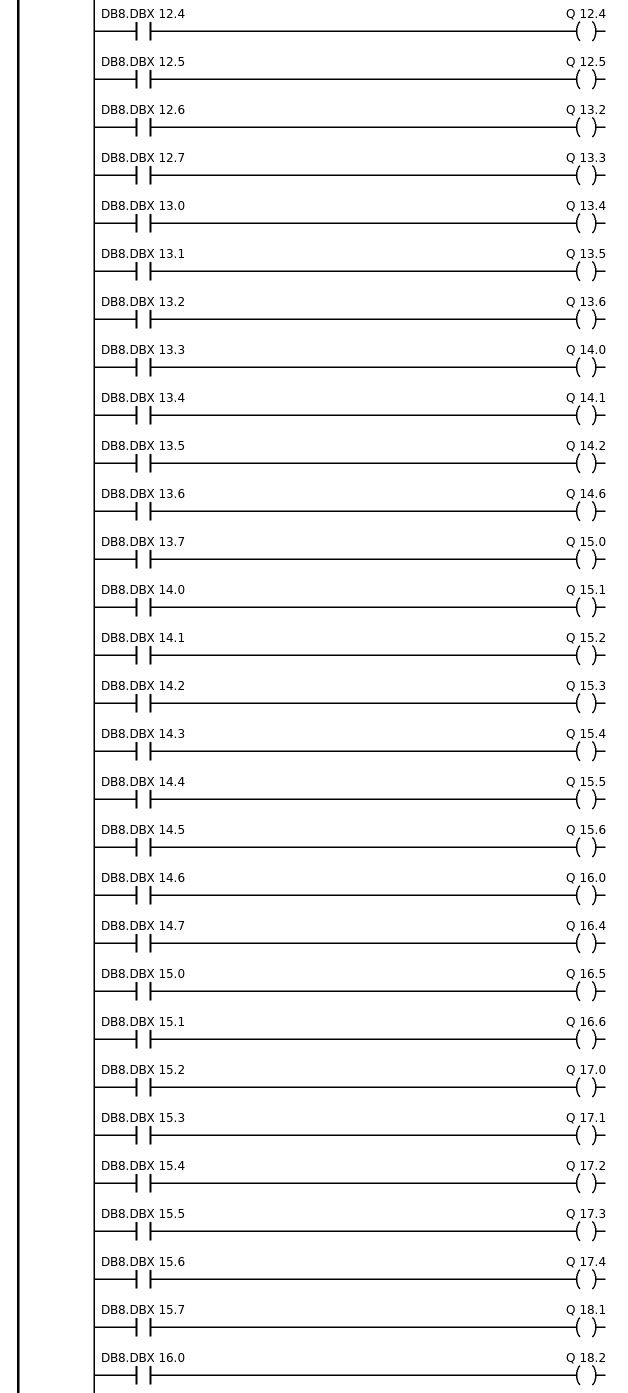
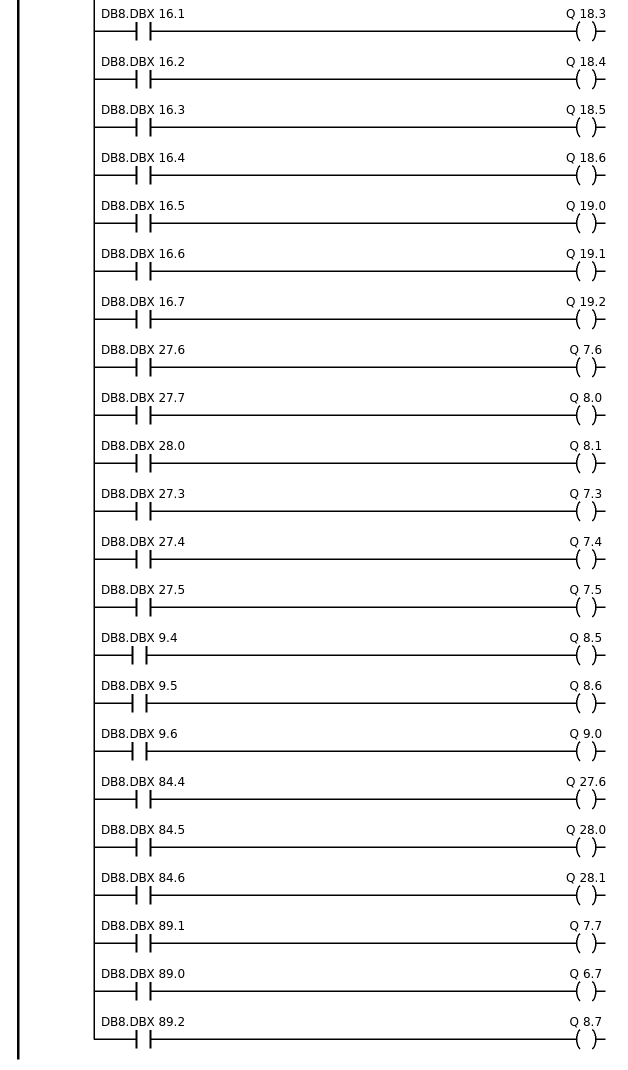
NETWORK
TITLE =
      A     M 0.1;
      =     L 0.0;
      A     L 0.0;
      A     DB8.DBX 26.7;
      =     Q 6.6;
      A     L 0.0;
      A     DB8.DBX 27.0;
      =     Q 7.0;
      A     L 0.0;
      A     DB8.DBX 27.1;
      =     Q 7.1;
      A     L 0.0;
      A     DB8.DBX 27.2;
      =     Q 7.2;
      A     L 0.0;
      A     DB8.DBX 9.1;
      =     Q 8.2;
      A     L 0.0;
      A     DB8.DBX 9.2;
      =     Q 8.3;
      A     L 0.0;
      A     DB8.DBX 9.3;
      =     Q 8.4;
      A     L 0.0;
      A     DB8.DBX 9.7;
      =     Q 9.1;
      A     L 0.0;
      A     DB8.DBX 10.0;
      =     Q 9.2;
      A     L 0.0;
      A     DB8.DBX 10.1;
      =     Q 9.3;
      A     L 0.0;
      A     DB8.DBX 10.2;
      =     Q 9.4;
      A     L 0.0;
      A     DB8.DBX 10.3;
      =     Q 9.5;
      A     L 0.0;
      A     DB8.DBX 10.4;
      =     Q 9.6;
      A     L 0.0;
      A     DB8.DBX 10.5;
      =     Q 10.0;
      A     L 0.0;
      A     DB8.DBX 10.6;
      =     Q 10.1;
      A     L 0.0;
      A     DB8.DBX 10.7;
      =     Q 10.2;
      A     L 0.0;
      A     DB8.DBX 11.0;
      =     Q 10.3;
      A     L 0.0;
      A     DB8.DBX 11.1;
      =     Q 10.4;
      A     L 0.0;
      A     DB8.DBX 11.2;
      =     Q 10.5;
      A     L 0.0;
      A     DB8.DBX 11.3;
      =     Q 10.6;
      A     L 0.0;
      A     DB8.DBX 11.4;
      =     Q 11.0;
      A     L 0.0;
      A     DB8.DBX 11.5;
      =     Q 11.4;
      A     L 0.0;
      A     DB8.DBX 11.6;
      =     Q 11.5;
      A     L 0.0;
      A     DB8.DBX 11.7;
      =     Q 11.6;
      A     L 0.0;
      A     DB8.DBX 12.0;
      =     Q 12.0;
      A     L 0.0;
      A     DB8.DBX 12.1;
      =     Q 12.1;
      A     L 0.0;
      A     DB8.DBX 12.2;
      =     Q 12.2;
      A     L 0.0;
      A     DB8.DBX 12.3;
      =     Q 12.3;
      A     L 0.0;
      A     DB8.DBX 12.4;
      =     Q 12.4;
      A     L 0.0;
      A     DB8.DBX 12.5;
      =     Q 12.5;
      A     L 0.0;
      A     DB8.DBX 12.6;
      =     Q 13.2;
      A     L 0.0;
      A     DB8.DBX 12.7;
      =     Q 13.3;
      A     L 0.0;
      A     DB8.DBX 13.0;
      =     Q 13.4;
      A     L 0.0;
      A     DB8.DBX 13.1;
      =     Q 13.5;
      A     L 0.0;
      A     DB8.DBX 13.2;
      =     Q 13.6;
      A     L 0.0;
      A     DB8.DBX 13.3;
      =     Q 14.0;
      A     L 0.0;
      A     DB8.DBX 13.4;
      =     Q 14.1;
      A     L 0.0;
      A     DB8.DBX 13.5;
      =     Q 14.2;
      A     L 0.0;
      A     DB8.DBX 13.6;
      =     Q 14.6;
      A     L 0.0;
      A     DB8.DBX 13.7;
      =     Q 15.0;
      A     L 0.0;
      A     DB8.DBX 14.0;
      =     Q 15.1;
      A     L 0.0;
      A     DB8.DBX 14.1;
      =     Q 15.2;
      A     L 0.0;
      A     DB8.DBX 14.2;
      =     Q 15.3;
      A     L 0.0;
      A     DB8.DBX 14.3;
      =     Q 15.4;
      A     L 0.0;
      A     DB8.DBX 14.4;
      =     Q 15.5;
      A     L 0.0;
      A     DB8.DBX 14.5;
      =     Q 15.6;
      A     L 0.0;
      A     DB8.DBX 14.6;
      =     Q 16.0;
      A     L 0.0;
      A     DB8.DBX 14.7;
      =     Q 16.4;
      A     L 0.0;
      A     DB8.DBX 15.0;
      =     Q 16.5;
      A     L 0.0;
      A     DB8.DBX 15.1;
      =     Q 16.6;
      A     L 0.0;
      A     DB8.DBX 15.2;
      =     Q 17.0;
      A     L 0.0;
      A     DB8.DBX 15.3;
      =     Q 17.1;
      A     L 0.0;
      A     DB8.DBX 15.4;
      =     Q 17.2;
      A     L 0.0;
      A     DB8.DBX 15.5;
      =     Q 17.3;
      A     L 0.0;
      A     DB8.DBX 15.6;
      =     Q 17.4;
      A     L 0.0;
      A     DB8.DBX 15.7;
      =     Q 18.1;
      A     L 0.0;
      A     DB8.DBX 16.0;
      =     Q 18.2;
      A     L 0.0;
      A     DB8.DBX 16.1;
      =     Q 18.3;
      A     L 0.0;
      A     DB8.DBX 16.2;
      =     Q 18.4;
      A     L 0.0;
      A     DB8.DBX 16.3;
      =     Q 18.5;
      A     L 0.0;
      A     DB8.DBX 16.4;
      =     Q 18.6;
      A     L 0.0;
      A     DB8.DBX 16.5;
      =     Q 19.0;
      A     L 0.0;
      A     DB8.DBX 16.6;
      =     Q 19.1;
      A     L 0.0;
      A     DB8.DBX 16.7;
      =     Q 19.2;
      A     L 0.0;
      A     DB8.DBX 27.6;
      =     Q 7.6;
      A     L 0.0;
      A     DB8.DBX 27.7;
      =     Q 8.0;
      A     L 0.0;
      A     DB8.DBX 28.0;
      =     Q 8.1;
      A     L 0.0;
      A     DB8.DBX 27.3;
      =     Q 7.3;
      A     L 0.0;
      A     DB8.DBX 27.4;
      =     Q 7.4;
      A     L 0.0;
      A     DB8.DBX 27.5;
      =     Q 7.5;
      A     L 0.0;
      A     DB8.DBX 9.4;
      =     Q 8.5;
      A     L 0.0;
      A     DB8.DBX 9.5;
      =     Q 8.6;
      A     L 0.0;
      A     DB8.DBX 9.6;
      =     Q 9.0;
      A     L 0.0;
      A     DB8.DBX 84.4;
      =     Q 27.6;
      A     L 0.0;
      A     DB8.DBX 84.5;
      =     Q 28.0;
      A     L 0.0;
      A     DB8.DBX 84.6;
      =     Q 28.1;
      A     L 0.0;
      A     DB8.DBX 89.1;
      =     Q 7.7;
      A     L 0.0;
      A     DB8.DBX 89.0;
      =     Q 6.7;
      A     L 0.0;
      A     DB8.DBX 89.2;
      =     Q 8.7;
END_FUNCTION

FUNCTION FC 7 : VOID
AUTHOR : Arun_Ram
VERSION : 0.1
BEGIN
// (block stored without names or comments; labels and parameter names are numbered)
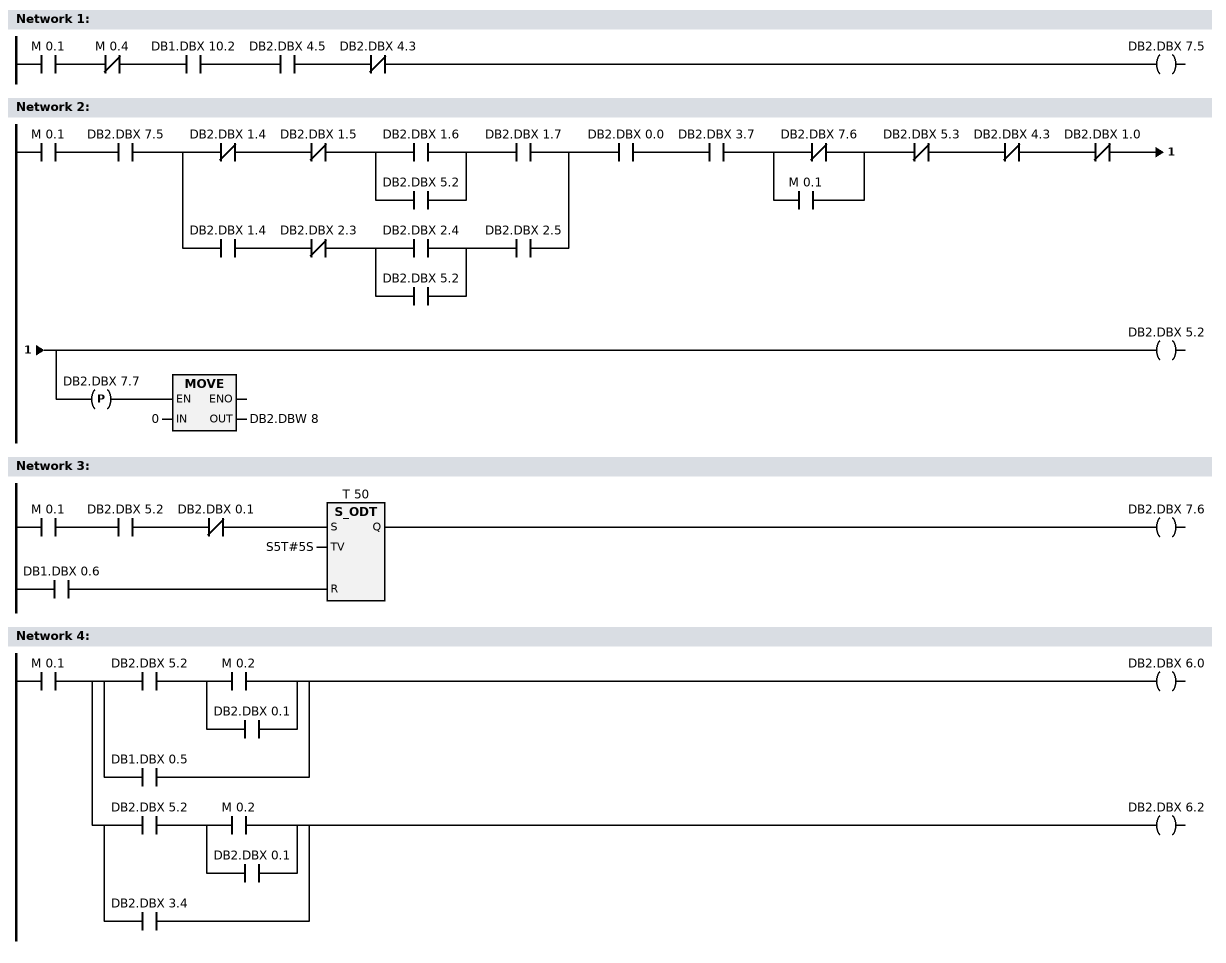
NETWORK
TITLE =
      A     M 0.1;
      AN    M 0.4;
      A     DB1.DBX 10.2;
      A     DB2.DBX 4.5;
      AN    DB2.DBX 4.3;
      =     DB2.DBX 7.5;
NETWORK
TITLE =
      A     M 0.1;
      A     DB2.DBX 7.5;
      A(;
      AN    DB2.DBX 1.4;
      AN    DB2.DBX 1.5;
      A(;
      O     DB2.DBX 1.6;
      O     DB2.DBX 5.2;
      );
      A     DB2.DBX 1.7;
      O;
      A     DB2.DBX 1.4;
      AN    DB2.DBX 2.3;
      A(;
      O     DB2.DBX 2.4;
      O     DB2.DBX 5.2;
      );
      A     DB2.DBX 2.5;
      );
      A     DB2.DBX 0.0;
      A     DB2.DBX 3.7;
      A(;
      ON    DB2.DBX 7.6;
      O     M 0.1;
      );
      AN    DB2.DBX 5.3;
      AN    DB2.DBX 4.3;
      AN    DB2.DBX 1.0;
      =     L 0.0;
      A     L 0.0;
      BLD   102;
      =     DB2.DBX 5.2;
      A     L 0.0;
      FP    DB2.DBX 7.7;
      JNB   M001;
      L     0;
      T     DB2.DBW 8;
M001: NOP   0;
NETWORK
TITLE =
      A     M 0.1;
      A     DB2.DBX 5.2;
      AN    DB2.DBX 0.1;
      L     S5T#5S;
      SD    T 50;
      A     DB1.DBX 0.6;
      R     T 50;
      NOP   0;
      NOP   0;
      A     T 50;
      =     DB2.DBX 7.6;
NETWORK
TITLE =
      A     M 0.1;
      =     L 0.0;
      A     L 0.0;
      A(;
      A     DB2.DBX 5.2;
      A(;
      O     M 0.2;
      O     DB2.DBX 0.1;
      );
      O     DB1.DBX 0.5;
      );
      =     DB2.DBX 6.0;
      A     L 0.0;
      A(;
      A     DB2.DBX 5.2;
      A(;
      O     M 0.2;
      O     DB2.DBX 0.1;
      );
      O     DB2.DBX 3.4;
      );
      =     DB2.DBX 6.2;
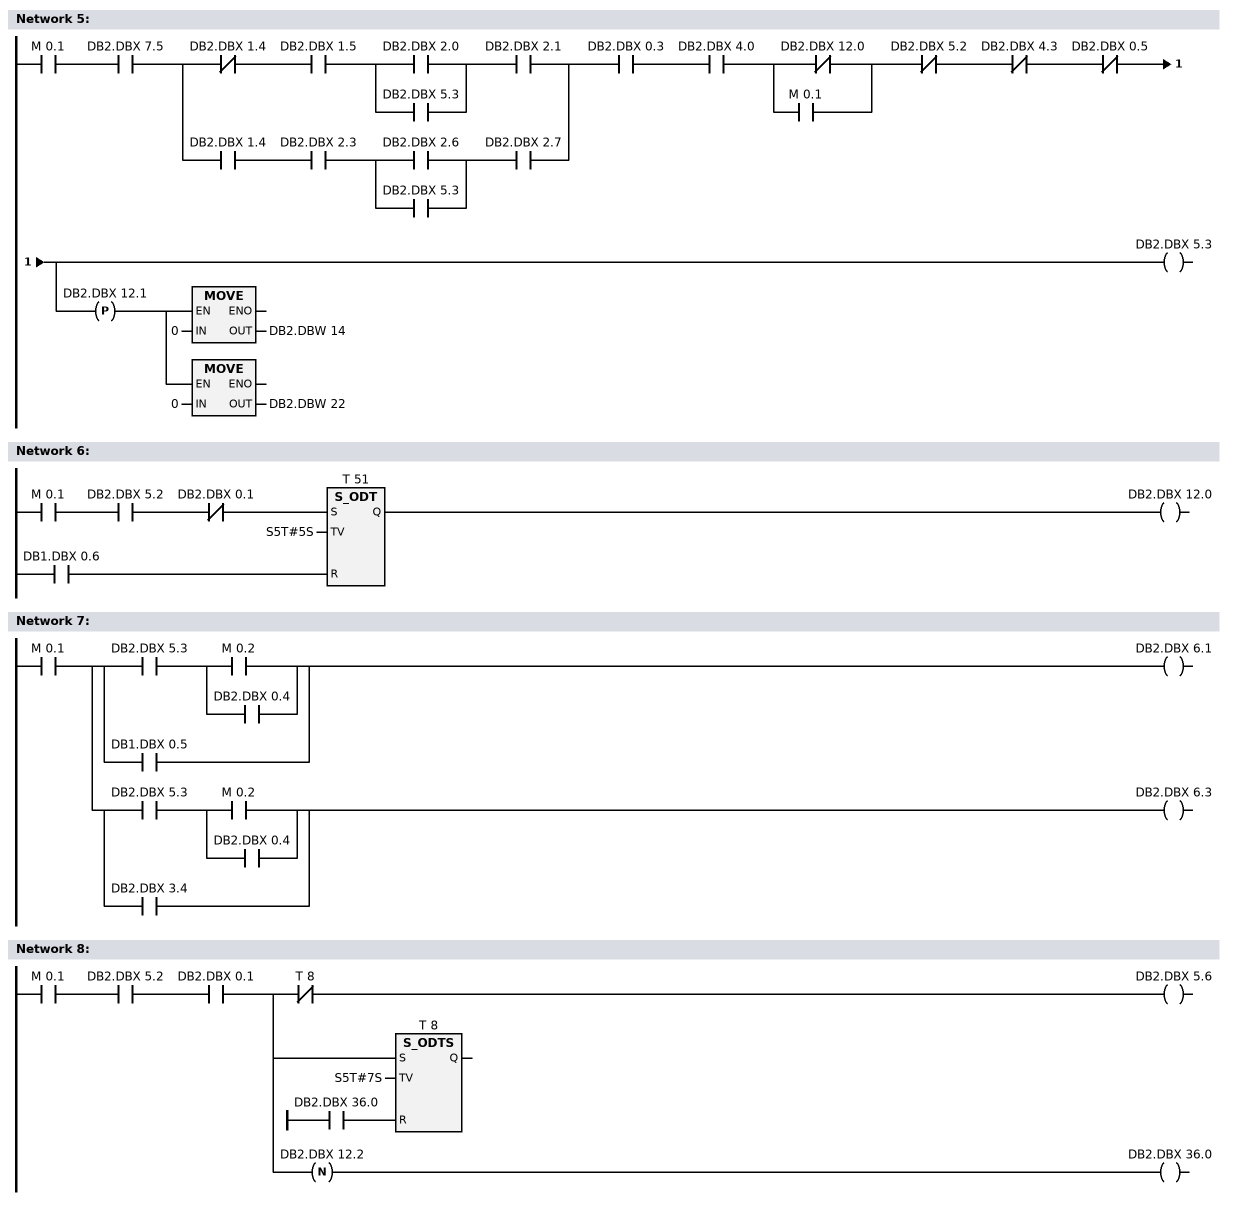
NETWORK
TITLE =
      A     M 0.1;
      A     DB2.DBX 7.5;
      A(;
      AN    DB2.DBX 1.4;
      A     DB2.DBX 1.5;
      A(;
      O     DB2.DBX 2.0;
      O     DB2.DBX 5.3;
      );
      A     DB2.DBX 2.1;
      O;
      A     DB2.DBX 1.4;
      A     DB2.DBX 2.3;
      A(;
      O     DB2.DBX 2.6;
      O     DB2.DBX 5.3;
      );
      A     DB2.DBX 2.7;
      );
      A     DB2.DBX 0.3;
      A     DB2.DBX 4.0;
      A(;
      ON    DB2.DBX 12.0;
      O     M 0.1;
      );
      AN    DB2.DBX 5.2;
      AN    DB2.DBX 4.3;
      AN    DB2.DBX 0.5;
      =     L 0.0;
      A     L 0.0;
      BLD   102;
      =     DB2.DBX 5.3;
      A     L 0.0;
      FP    DB2.DBX 12.1;
      =     L 0.1;
      A     L 0.1;
      JNB   M002;
      L     0;
      T     DB2.DBW 14;
M002: NOP   0;
      A     L 0.1;
      JNB   M003;
      L     0;
      T     DB2.DBW 22;
M003: NOP   0;
NETWORK
TITLE =
      A     M 0.1;
      A     DB2.DBX 5.2;
      AN    DB2.DBX 0.1;
      L     S5T#5S;
      SD    T 51;
      A     DB1.DBX 0.6;
      R     T 51;
      NOP   0;
      NOP   0;
      A     T 51;
      =     DB2.DBX 12.0;
NETWORK
TITLE =
      A     M 0.1;
      =     L 0.0;
      A     L 0.0;
      A(;
      A     DB2.DBX 5.3;
      A(;
      O     M 0.2;
      O     DB2.DBX 0.4;
      );
      O     DB1.DBX 0.5;
      );
      =     DB2.DBX 6.1;
      A     L 0.0;
      A(;
      A     DB2.DBX 5.3;
      A(;
      O     M 0.2;
      O     DB2.DBX 0.4;
      );
      O     DB2.DBX 3.4;
      );
      =     DB2.DBX 6.3;
NETWORK
TITLE =
      A     M 0.1;
      A     DB2.DBX 5.2;
      A     DB2.DBX 0.1;
      =     L 0.0;
      A     L 0.0;
      AN    T 8;
      =     DB2.DBX 5.6;
      A     L 0.0;
      L     S5T#7S;
      SS    T 8;
      A     DB2.DBX 36.0;
      R     T 8;
      NOP   0;
      NOP   0;
      NOP   0;
      A     L 0.0;
      FN    DB2.DBX 12.2;
      =     DB2.DBX 36.0;
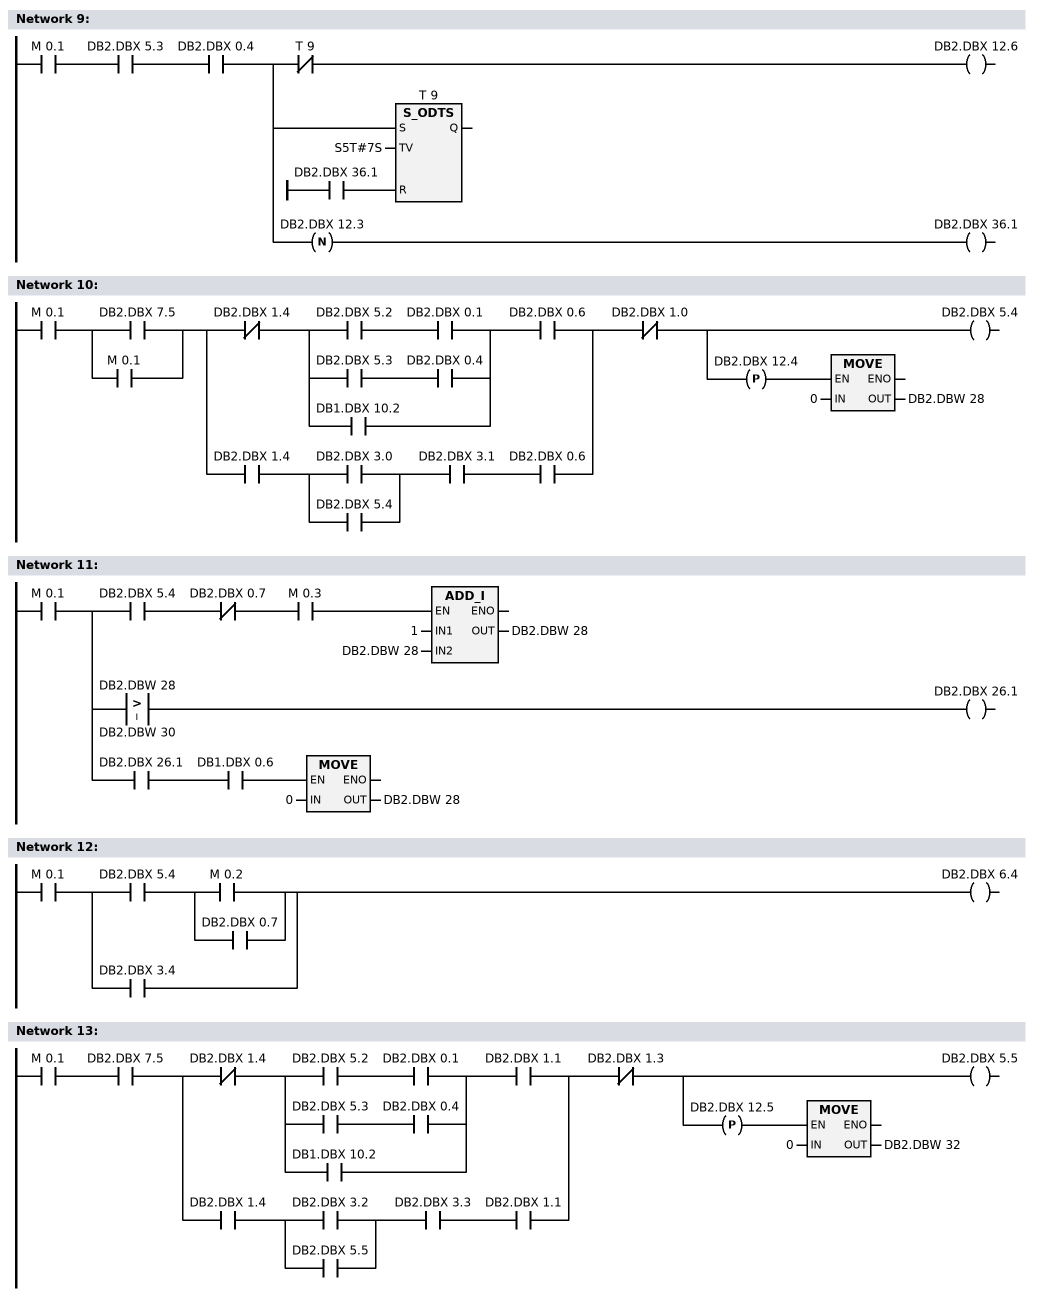
NETWORK
TITLE =
      A     M 0.1;
      A     DB2.DBX 5.3;
      A     DB2.DBX 0.4;
      =     L 0.0;
      A     L 0.0;
      AN    T 9;
      =     DB2.DBX 12.6;
      A     L 0.0;
      L     S5T#7S;
      SS    T 9;
      A     DB2.DBX 36.1;
      R     T 9;
      NOP   0;
      NOP   0;
      NOP   0;
      A     L 0.0;
      FN    DB2.DBX 12.3;
      =     DB2.DBX 36.1;
NETWORK
TITLE =
      A     M 0.1;
      A(;
      O     DB2.DBX 7.5;
      O     M 0.1;
      );
      A(;
      AN    DB2.DBX 1.4;
      A(;
      A     DB2.DBX 5.2;
      A     DB2.DBX 0.1;
      O;
      A     DB2.DBX 5.3;
      A     DB2.DBX 0.4;
      O     DB1.DBX 10.2;
      );
      A     DB2.DBX 0.6;
      O;
      A     DB2.DBX 1.4;
      A(;
      O     DB2.DBX 3.0;
      O     DB2.DBX 5.4;
      );
      A     DB2.DBX 3.1;
      A     DB2.DBX 0.6;
      );
      AN    DB2.DBX 1.0;
      =     L 0.0;
      A     L 0.0;
      BLD   102;
      =     DB2.DBX 5.4;
      A     L 0.0;
      FP    DB2.DBX 12.4;
      JNB   M004;
      L     0;
      T     DB2.DBW 28;
M004: NOP   0;
NETWORK
TITLE =
      A     M 0.1;
      =     L 0.0;
      A     L 0.0;
      A     DB2.DBX 5.4;
      AN    DB2.DBX 0.7;
      A     M 0.3;
      JNB   M005;
      L     1;
      L     DB2.DBW 28;
      +I;
      T     DB2.DBW 28;
M005: NOP   0;
      A     L 0.0;
      A(;
      L     DB2.DBW 28;
      L     DB2.DBW 30;
      >I;
      );
      =     DB2.DBX 26.1;
      A     L 0.0;
      A     DB2.DBX 26.1;
      A     DB1.DBX 0.6;
      JNB   M006;
      L     0;
      T     DB2.DBW 28;
M006: NOP   0;
NETWORK
TITLE =
      A     M 0.1;
      A(;
      A     DB2.DBX 5.4;
      A(;
      O     M 0.2;
      O     DB2.DBX 0.7;
      );
      O     DB2.DBX 3.4;
      );
      =     DB2.DBX 6.4;
NETWORK
TITLE =
      A     M 0.1;
      A     DB2.DBX 7.5;
      A(;
      AN    DB2.DBX 1.4;
      A(;
      A     DB2.DBX 5.2;
      A     DB2.DBX 0.1;
      O;
      A     DB2.DBX 5.3;
      A     DB2.DBX 0.4;
      O     DB1.DBX 10.2;
      );
      A     DB2.DBX 1.1;
      O;
      A     DB2.DBX 1.4;
      A(;
      O     DB2.DBX 3.2;
      O     DB2.DBX 5.5;
      );
      A     DB2.DBX 3.3;
      A     DB2.DBX 1.1;
      );
      AN    DB2.DBX 1.3;
      =     L 0.0;
      A     L 0.0;
      BLD   102;
      =     DB2.DBX 5.5;
      A     L 0.0;
      FP    DB2.DBX 12.5;
      JNB   M007;
      L     0;
      T     DB2.DBW 32;
M007: NOP   0;
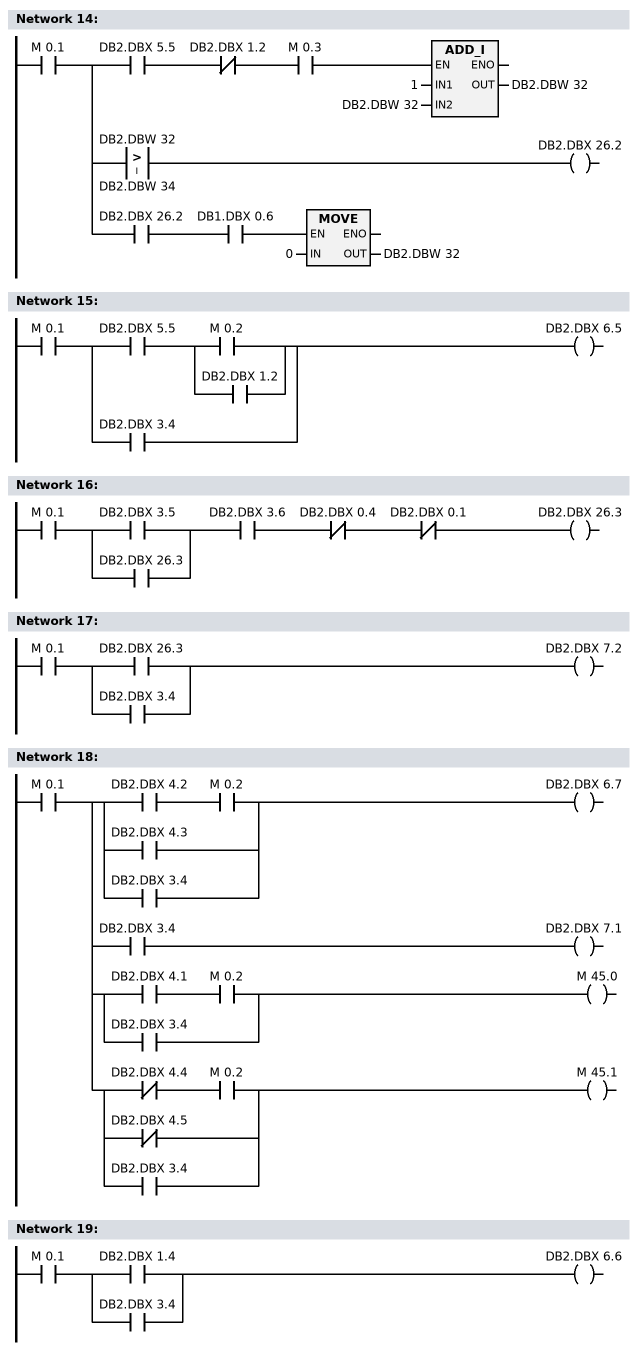
NETWORK
TITLE =
      A     M 0.1;
      =     L 0.0;
      A     L 0.0;
      A     DB2.DBX 5.5;
      AN    DB2.DBX 1.2;
      A     M 0.3;
      JNB   M008;
      L     1;
      L     DB2.DBW 32;
      +I;
      T     DB2.DBW 32;
M008: NOP   0;
      A     L 0.0;
      A(;
      L     DB2.DBW 32;
      L     DB2.DBW 34;
      >I;
      );
      =     DB2.DBX 26.2;
      A     L 0.0;
      A     DB2.DBX 26.2;
      A     DB1.DBX 0.6;
      JNB   M009;
      L     0;
      T     DB2.DBW 32;
M009: NOP   0;
NETWORK
TITLE =
      A     M 0.1;
      A(;
      A     DB2.DBX 5.5;
      A(;
      O     M 0.2;
      O     DB2.DBX 1.2;
      );
      O     DB2.DBX 3.4;
      );
      =     DB2.DBX 6.5;
NETWORK
TITLE =
      A     M 0.1;
      A(;
      O     DB2.DBX 3.5;
      O     DB2.DBX 26.3;
      );
      A     DB2.DBX 3.6;
      AN    DB2.DBX 0.4;
      AN    DB2.DBX 0.1;
      =     DB2.DBX 26.3;
NETWORK
TITLE =
      A     M 0.1;
      A(;
      O     DB2.DBX 26.3;
      O     DB2.DBX 3.4;
      );
      =     DB2.DBX 7.2;
NETWORK
TITLE =
      A     M 0.1;
      =     L 0.0;
      A     L 0.0;
      A(;
      A     DB2.DBX 4.2;
      A     M 0.2;
      O     DB2.DBX 4.3;
      O     DB2.DBX 3.4;
      );
      =     DB2.DBX 6.7;
      A     L 0.0;
      A     DB2.DBX 3.4;
      =     DB2.DBX 7.1;
      A     L 0.0;
      A(;
      A     DB2.DBX 4.1;
      A     M 0.2;
      O     DB2.DBX 3.4;
      );
      =     M 45.0;
      A     L 0.0;
      A(;
      AN    DB2.DBX 4.4;
      A     M 0.2;
      ON    DB2.DBX 4.5;
      O     DB2.DBX 3.4;
      );
      =     M 45.1;
NETWORK
TITLE =
      A     M 0.1;
      A(;
      O     DB2.DBX 1.4;
      O     DB2.DBX 3.4;
      );
      =     DB2.DBX 6.6;
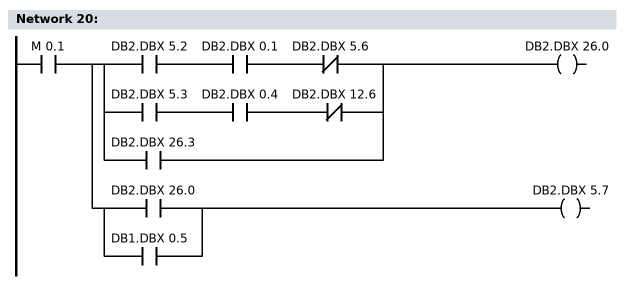
NETWORK
TITLE =
      A     M 0.1;
      =     L 0.0;
      A     L 0.0;
      A(;
      A     DB2.DBX 5.2;
      A     DB2.DBX 0.1;
      AN    DB2.DBX 5.6;
      O;
      A     DB2.DBX 5.3;
      A     DB2.DBX 0.4;
      AN    DB2.DBX 12.6;
      O     DB2.DBX 26.3;
      );
      =     DB2.DBX 26.0;
      A     L 0.0;
      A(;
      O     DB2.DBX 26.0;
      O     DB1.DBX 0.5;
      );
      =     DB2.DBX 5.7;
END_FUNCTION

FUNCTION FC 8 : VOID
AUTHOR : Arun_Ram
VERSION : 0.1
BEGIN
// (block stored without names or comments; labels and parameter names are numbered)
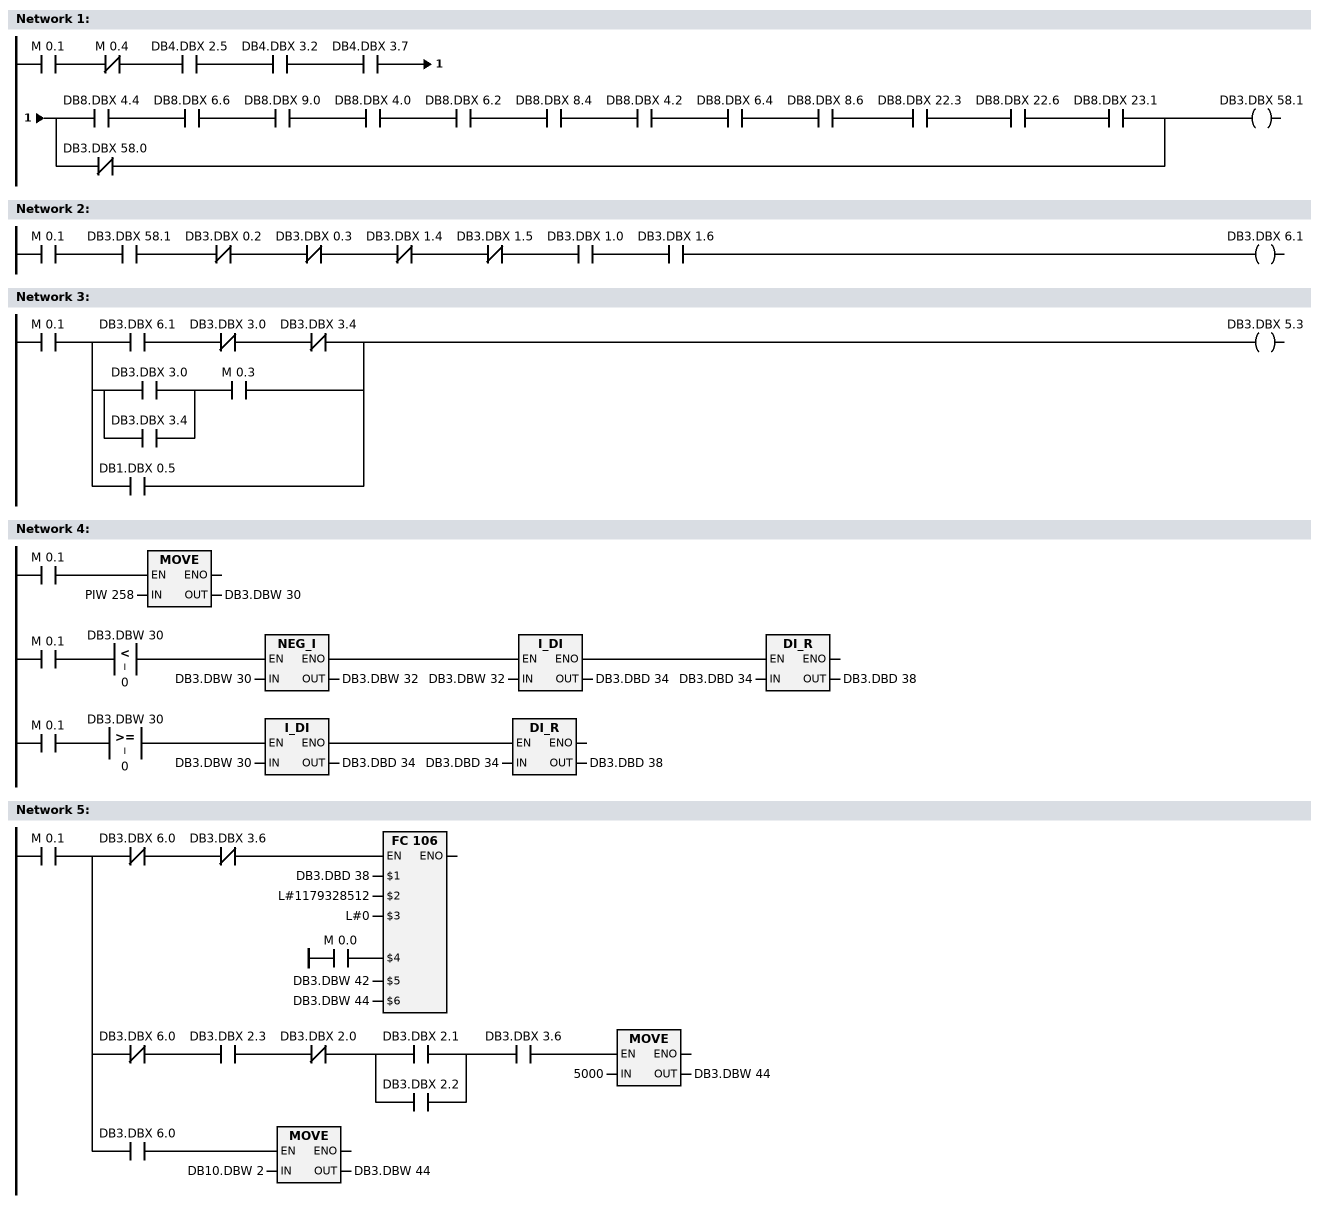
NETWORK
TITLE =
      A     M 0.1;
      AN    M 0.4;
      A     DB4.DBX 2.5;
      A     DB4.DBX 3.2;
      A     DB4.DBX 3.7;
      A(;
      A     DB8.DBX 4.4;
      A     DB8.DBX 6.6;
      A     DB8.DBX 9.0;
      A     DB8.DBX 4.0;
      A     DB8.DBX 6.2;
      A     DB8.DBX 8.4;
      A     DB8.DBX 4.2;
      A     DB8.DBX 6.4;
      A     DB8.DBX 8.6;
      A     DB8.DBX 22.3;
      A     DB8.DBX 22.6;
      A     DB8.DBX 23.1;
      ON    DB3.DBX 58.0;
      );
      =     DB3.DBX 58.1;
NETWORK
TITLE =
      A     M 0.1;
      A     DB3.DBX 58.1;
      AN    DB3.DBX 0.2;
      AN    DB3.DBX 0.3;
      AN    DB3.DBX 1.4;
      AN    DB3.DBX 1.5;
      A     DB3.DBX 1.0;
      A     DB3.DBX 1.6;
      =     DB3.DBX 6.1;
NETWORK
TITLE =
      A     M 0.1;
      A(;
      A     DB3.DBX 6.1;
      AN    DB3.DBX 3.0;
      AN    DB3.DBX 3.4;
      O;
      A(;
      O     DB3.DBX 3.0;
      O     DB3.DBX 3.4;
      );
      A     M 0.3;
      O     DB1.DBX 0.5;
      );
      =     DB3.DBX 5.3;
NETWORK
TITLE =
      A     M 0.1;
      =     L 0.0;
      A     L 0.0;
      JNB   M001;
      L     PIW 258;
      T     DB3.DBW 30;
M001: NOP   0;
      A(;
      A(;
      A     L 0.0;
      A(;
      L     DB3.DBW 30;
      L     0;
      <I;
      );
      JNB   M002;
      L     DB3.DBW 30;
      NEGI;
      T     DB3.DBW 32;
      AN    OV;
      SAVE;
      CLR;
M002: A     BR;
      );
      JNB   M003;
      L     DB3.DBW 32;
      ITD;
      T     DB3.DBD 34;
      SET;
      SAVE;
      CLR;
M003: A     BR;
      );
      JNB   M004;
      L     DB3.DBD 34;
      DTR;
      T     DB3.DBD 38;
M004: NOP   0;
      A(;
      A     L 0.0;
      A(;
      L     DB3.DBW 30;
      L     0;
      >=I;
      );
      JNB   M005;
      L     DB3.DBW 30;
      ITD;
      T     DB3.DBD 34;
      SET;
      SAVE;
      CLR;
M005: A     BR;
      );
      JNB   M006;
      L     DB3.DBD 34;
      DTR;
      T     DB3.DBD 38;
M006: NOP   0;
NETWORK
TITLE =
      A     M 0.1;
      =     L 0.0;
      A     M 0.0;
      =     L 0.1;
      BLD   103;
      A     L 0.0;
      AN    DB3.DBX 6.0;
      AN    DB3.DBX 3.6;
      JNB   M007;
      CALL  FC 106 (
           $1                       := DB3.DBD 38,
           $2                       := L#1179328512,
           $3                       := L#0,
           $4                       := L 0.1,
           $5                       := DB3.DBW 42,
           $6                       := DB3.DBW 44);
M007: NOP   0;
      A     L 0.0;
      AN    DB3.DBX 6.0;
      A     DB3.DBX 2.3;
      AN    DB3.DBX 2.0;
      A(;
      O     DB3.DBX 2.1;
      O     DB3.DBX 2.2;
      );
      A     DB3.DBX 3.6;
      JNB   M008;
      L     5000;
      T     DB3.DBW 44;
M008: NOP   0;
      A     L 0.0;
      A     DB3.DBX 6.0;
      JNB   M009;
      L     DB10.DBW 2;
      T     DB3.DBW 44;
M009: NOP   0;
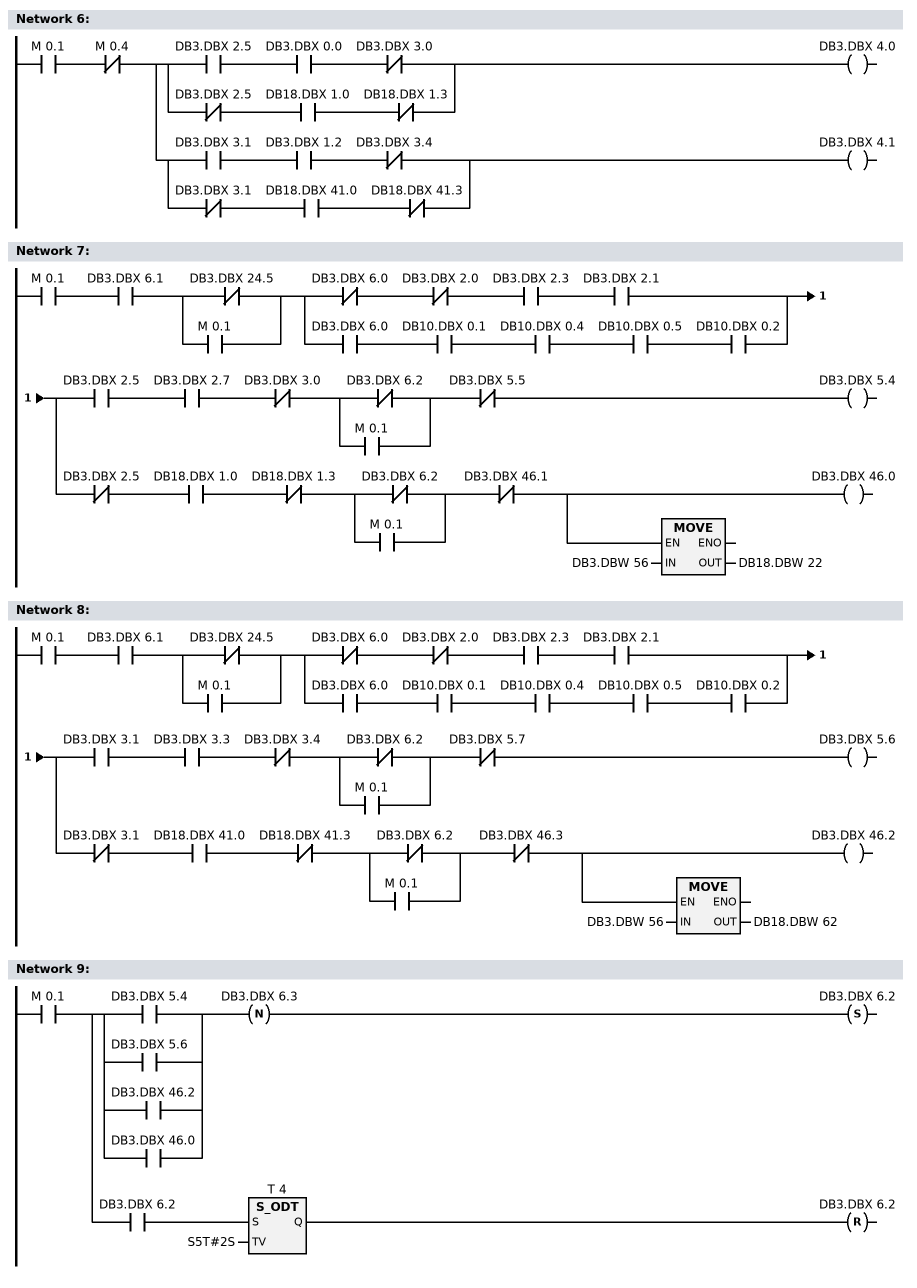
NETWORK
TITLE =
      A     M 0.1;
      AN    M 0.4;
      =     L 0.0;
      A     L 0.0;
      A(;
      A     DB3.DBX 2.5;
      A     DB3.DBX 0.0;
      AN    DB3.DBX 3.0;
      O;
      AN    DB3.DBX 2.5;
      A     DB18.DBX 1.0;
      AN    DB18.DBX 1.3;
      );
      =     DB3.DBX 4.0;
      A     L 0.0;
      A(;
      A     DB3.DBX 3.1;
      A     DB3.DBX 1.2;
      AN    DB3.DBX 3.4;
      O;
      AN    DB3.DBX 3.1;
      A     DB18.DBX 41.0;
      AN    DB18.DBX 41.3;
      );
      =     DB3.DBX 4.1;
NETWORK
TITLE =
      A     M 0.1;
      A     DB3.DBX 6.1;
      A(;
      ON    DB3.DBX 24.5;
      O     M 0.1;
      );
      A(;
      AN    DB3.DBX 6.0;
      AN    DB3.DBX 2.0;
      A     DB3.DBX 2.3;
      A     DB3.DBX 2.1;
      O;
      A     DB3.DBX 6.0;
      A     DB10.DBX 0.1;
      A     DB10.DBX 0.4;
      A     DB10.DBX 0.5;
      A     DB10.DBX 0.2;
      );
      =     L 0.0;
      A     L 0.0;
      A     DB3.DBX 2.5;
      A     DB3.DBX 2.7;
      AN    DB3.DBX 3.0;
      A(;
      ON    DB3.DBX 6.2;
      O     M 0.1;
      );
      AN    DB3.DBX 5.5;
      =     DB3.DBX 5.4;
      A     L 0.0;
      AN    DB3.DBX 2.5;
      A     DB18.DBX 1.0;
      AN    DB18.DBX 1.3;
      A(;
      ON    DB3.DBX 6.2;
      O     M 0.1;
      );
      AN    DB3.DBX 46.1;
      =     L 0.1;
      A     L 0.1;
      BLD   102;
      =     DB3.DBX 46.0;
      A     L 0.1;
      JNB   M010;
      L     DB3.DBW 56;
      T     DB18.DBW 22;
M010: NOP   0;
NETWORK
TITLE =
      A     M 0.1;
      A     DB3.DBX 6.1;
      A(;
      ON    DB3.DBX 24.5;
      O     M 0.1;
      );
      A(;
      AN    DB3.DBX 6.0;
      AN    DB3.DBX 2.0;
      A     DB3.DBX 2.3;
      A     DB3.DBX 2.1;
      O;
      A     DB3.DBX 6.0;
      A     DB10.DBX 0.1;
      A     DB10.DBX 0.4;
      A     DB10.DBX 0.5;
      A     DB10.DBX 0.2;
      );
      =     L 0.0;
      A     L 0.0;
      A     DB3.DBX 3.1;
      A     DB3.DBX 3.3;
      AN    DB3.DBX 3.4;
      A(;
      ON    DB3.DBX 6.2;
      O     M 0.1;
      );
      AN    DB3.DBX 5.7;
      =     DB3.DBX 5.6;
      A     L 0.0;
      AN    DB3.DBX 3.1;
      A     DB18.DBX 41.0;
      AN    DB18.DBX 41.3;
      A(;
      ON    DB3.DBX 6.2;
      O     M 0.1;
      );
      AN    DB3.DBX 46.3;
      =     L 0.1;
      A     L 0.1;
      BLD   102;
      =     DB3.DBX 46.2;
      A     L 0.1;
      JNB   M011;
      L     DB3.DBW 56;
      T     DB18.DBW 62;
M011: NOP   0;
NETWORK
TITLE =
      A     M 0.1;
      =     L 0.0;
      A     L 0.0;
      A(;
      O     DB3.DBX 5.4;
      O     DB3.DBX 5.6;
      O     DB3.DBX 46.2;
      O     DB3.DBX 46.0;
      );
      FN    DB3.DBX 6.3;
      S     DB3.DBX 6.2;
      A     L 0.0;
      A     DB3.DBX 6.2;
      L     S5T#2S;
      SD    T 4;
      NOP   0;
      NOP   0;
      NOP   0;
      A     T 4;
      R     DB3.DBX 6.2;
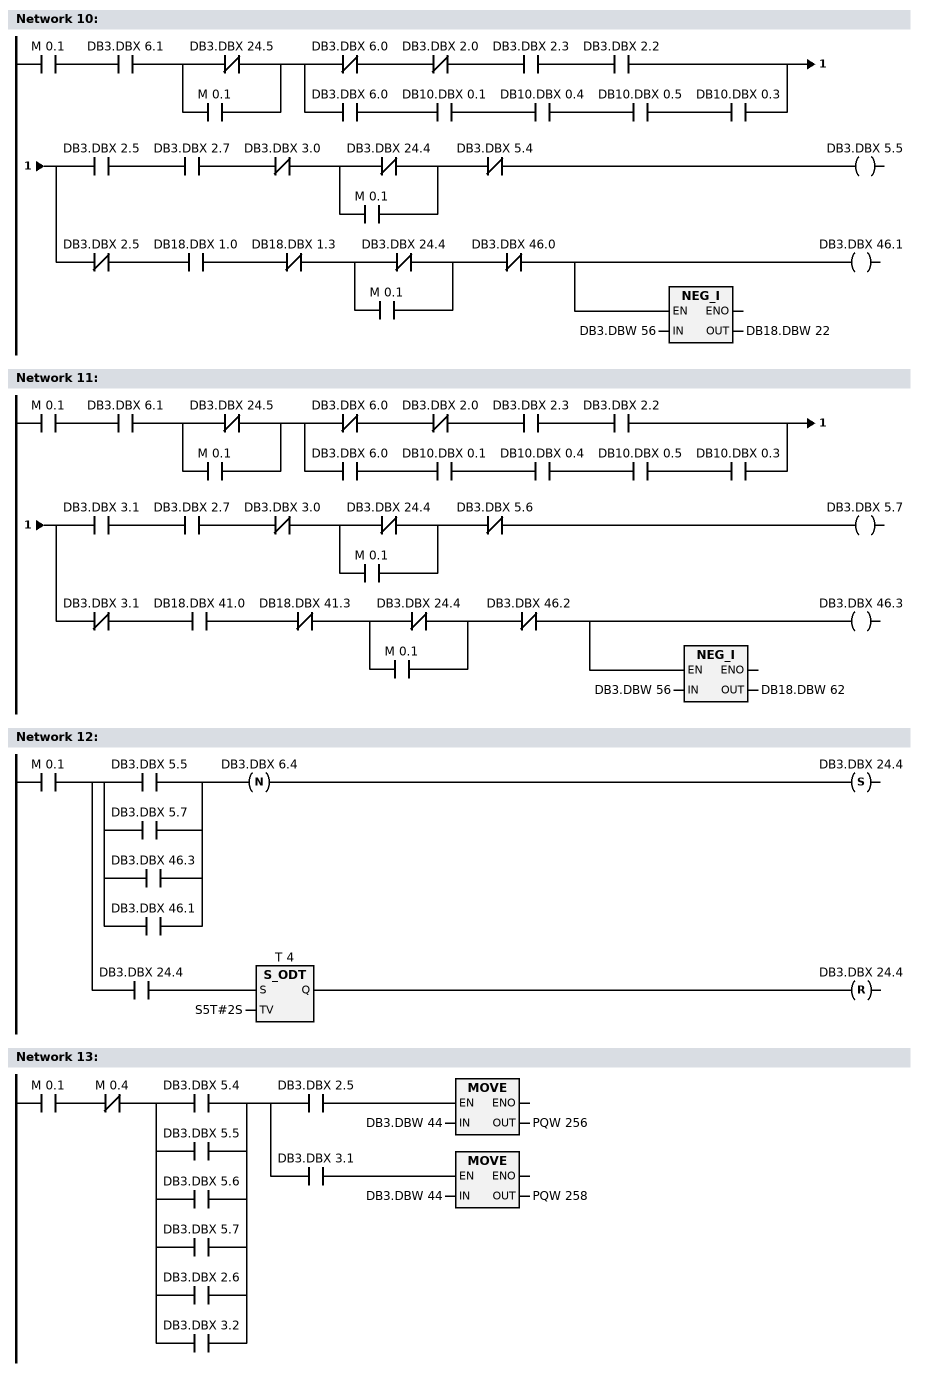
NETWORK
TITLE =
      A     M 0.1;
      A     DB3.DBX 6.1;
      A(;
      ON    DB3.DBX 24.5;
      O     M 0.1;
      );
      A(;
      AN    DB3.DBX 6.0;
      AN    DB3.DBX 2.0;
      A     DB3.DBX 2.3;
      A     DB3.DBX 2.2;
      O;
      A     DB3.DBX 6.0;
      A     DB10.DBX 0.1;
      A     DB10.DBX 0.4;
      A     DB10.DBX 0.5;
      A     DB10.DBX 0.3;
      );
      =     L 0.0;
      A     L 0.0;
      A     DB3.DBX 2.5;
      A     DB3.DBX 2.7;
      AN    DB3.DBX 3.0;
      A(;
      ON    DB3.DBX 24.4;
      O     M 0.1;
      );
      AN    DB3.DBX 5.4;
      =     DB3.DBX 5.5;
      A     L 0.0;
      AN    DB3.DBX 2.5;
      A     DB18.DBX 1.0;
      AN    DB18.DBX 1.3;
      A(;
      ON    DB3.DBX 24.4;
      O     M 0.1;
      );
      AN    DB3.DBX 46.0;
      =     L 0.1;
      A     L 0.1;
      BLD   102;
      =     DB3.DBX 46.1;
      A     L 0.1;
      JNB   M012;
      L     DB3.DBW 56;
      NEGI;
      T     DB18.DBW 22;
M012: NOP   0;
NETWORK
TITLE =
      A     M 0.1;
      A     DB3.DBX 6.1;
      A(;
      ON    DB3.DBX 24.5;
      O     M 0.1;
      );
      A(;
      AN    DB3.DBX 6.0;
      AN    DB3.DBX 2.0;
      A     DB3.DBX 2.3;
      A     DB3.DBX 2.2;
      O;
      A     DB3.DBX 6.0;
      A     DB10.DBX 0.1;
      A     DB10.DBX 0.4;
      A     DB10.DBX 0.5;
      A     DB10.DBX 0.3;
      );
      =     L 0.0;
      A     L 0.0;
      A     DB3.DBX 3.1;
      A     DB3.DBX 2.7;
      AN    DB3.DBX 3.0;
      A(;
      ON    DB3.DBX 24.4;
      O     M 0.1;
      );
      AN    DB3.DBX 5.6;
      =     DB3.DBX 5.7;
      A     L 0.0;
      AN    DB3.DBX 3.1;
      A     DB18.DBX 41.0;
      AN    DB18.DBX 41.3;
      A(;
      ON    DB3.DBX 24.4;
      O     M 0.1;
      );
      AN    DB3.DBX 46.2;
      =     L 0.1;
      A     L 0.1;
      BLD   102;
      =     DB3.DBX 46.3;
      A     L 0.1;
      JNB   M013;
      L     DB3.DBW 56;
      NEGI;
      T     DB18.DBW 62;
M013: NOP   0;
NETWORK
TITLE =
      A     M 0.1;
      =     L 0.0;
      A     L 0.0;
      A(;
      O     DB3.DBX 5.5;
      O     DB3.DBX 5.7;
      O     DB3.DBX 46.3;
      O     DB3.DBX 46.1;
      );
      FN    DB3.DBX 6.4;
      S     DB3.DBX 24.4;
      A     L 0.0;
      A     DB3.DBX 24.4;
      L     S5T#2S;
      SD    T 4;
      NOP   0;
      NOP   0;
      NOP   0;
      A     T 4;
      R     DB3.DBX 24.4;
NETWORK
TITLE =
      A     M 0.1;
      AN    M 0.4;
      A(;
      O     DB3.DBX 5.4;
      O     DB3.DBX 5.5;
      O     DB3.DBX 5.6;
      O     DB3.DBX 5.7;
      O     DB3.DBX 2.6;
      O     DB3.DBX 3.2;
      );
      =     L 0.0;
      A     L 0.0;
      A     DB3.DBX 2.5;
      JNB   M014;
      L     DB3.DBW 44;
      T     PQW 256;
M014: NOP   0;
      A     L 0.0;
      A     DB3.DBX 3.1;
      JNB   M015;
      L     DB3.DBW 44;
      T     PQW 258;
M015: NOP   0;
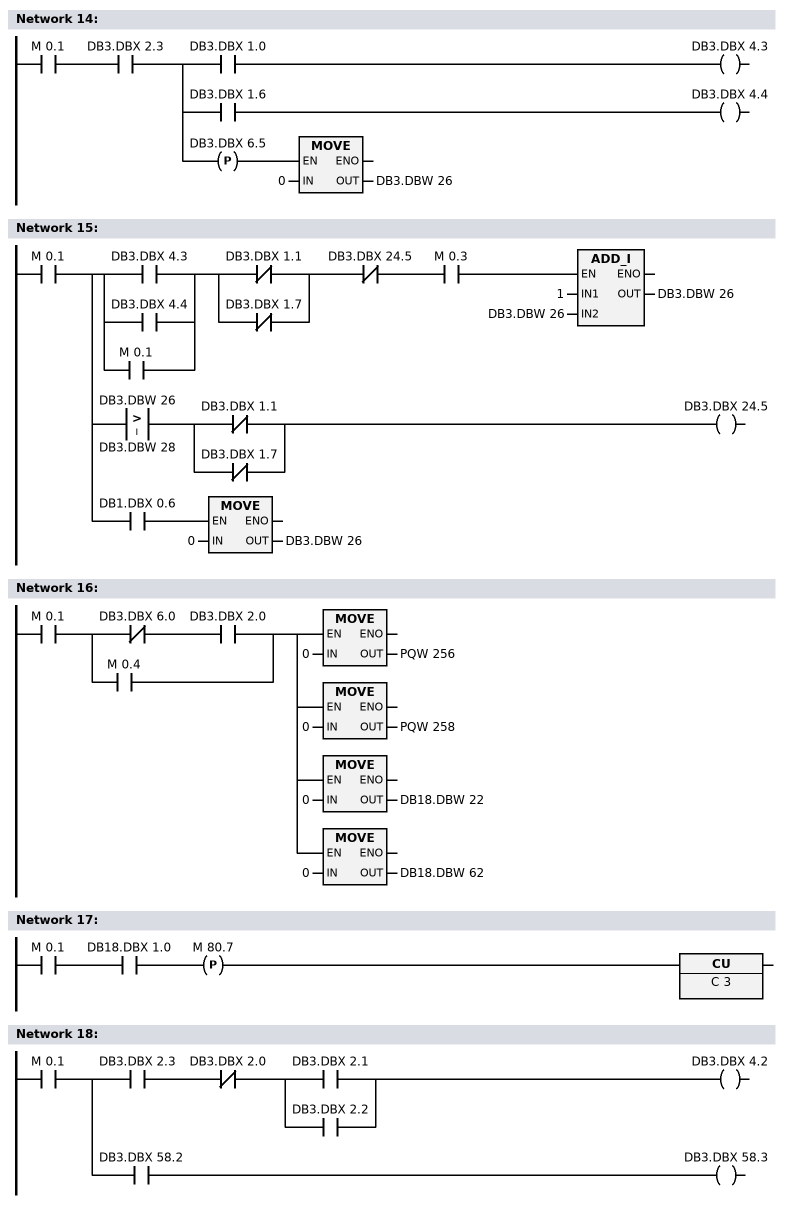
NETWORK
TITLE =
      A     M 0.1;
      A     DB3.DBX 2.3;
      =     L 0.0;
      A     L 0.0;
      A     DB3.DBX 1.0;
      =     DB3.DBX 4.3;
      A     L 0.0;
      A     DB3.DBX 1.6;
      =     DB3.DBX 4.4;
      A     L 0.0;
      FP    DB3.DBX 6.5;
      JNB   M016;
      L     0;
      T     DB3.DBW 26;
M016: NOP   0;
NETWORK
TITLE =
      A     M 0.1;
      =     L 0.0;
      A     L 0.0;
      A(;
      O     DB3.DBX 4.3;
      O     DB3.DBX 4.4;
      O     M 0.1;
      );
      A(;
      ON    DB3.DBX 1.1;
      ON    DB3.DBX 1.7;
      );
      AN    DB3.DBX 24.5;
      A     M 0.3;
      JNB   M017;
      L     1;
      L     DB3.DBW 26;
      +I;
      T     DB3.DBW 26;
M017: NOP   0;
      A     L 0.0;
      A(;
      L     DB3.DBW 26;
      L     DB3.DBW 28;
      >I;
      );
      A(;
      ON    DB3.DBX 1.1;
      ON    DB3.DBX 1.7;
      );
      =     DB3.DBX 24.5;
      A     L 0.0;
      A     DB1.DBX 0.6;
      JNB   M018;
      L     0;
      T     DB3.DBW 26;
M018: NOP   0;
NETWORK
TITLE =
      A     M 0.1;
      A(;
      AN    DB3.DBX 6.0;
      A     DB3.DBX 2.0;
      O     M 0.4;
      );
      =     L 0.0;
      A     L 0.0;
      JNB   M019;
      L     0;
      T     PQW 256;
M019: NOP   0;
      A     L 0.0;
      JNB   M020;
      L     0;
      T     PQW 258;
M020: NOP   0;
      A     L 0.0;
      JNB   M021;
      L     0;
      T     DB18.DBW 22;
M021: NOP   0;
      A     L 0.0;
      JNB   M022;
      L     0;
      T     DB18.DBW 62;
M022: NOP   0;
NETWORK
TITLE =
      A     M 0.1;
      A     DB18.DBX 1.0;
      FP    M 80.7;
      CU    C 3;
      BLD   101;
      NOP   0;
      NOP   0;
      NOP   0;
      NOP   0;
      NOP   0;
      NOP   0;
NETWORK
TITLE =
      A     M 0.1;
      =     L 0.0;
      A     L 0.0;
      A     DB3.DBX 2.3;
      AN    DB3.DBX 2.0;
      A(;
      O     DB3.DBX 2.1;
      O     DB3.DBX 2.2;
      );
      =     DB3.DBX 4.2;
      A     L 0.0;
      A     DB3.DBX 58.2;
      =     DB3.DBX 58.3;
END_FUNCTION

FUNCTION FC 9 : VOID
AUTHOR : Arun
VERSION : 0.1
BEGIN
// (block stored without names or comments; labels and parameter names are numbered)
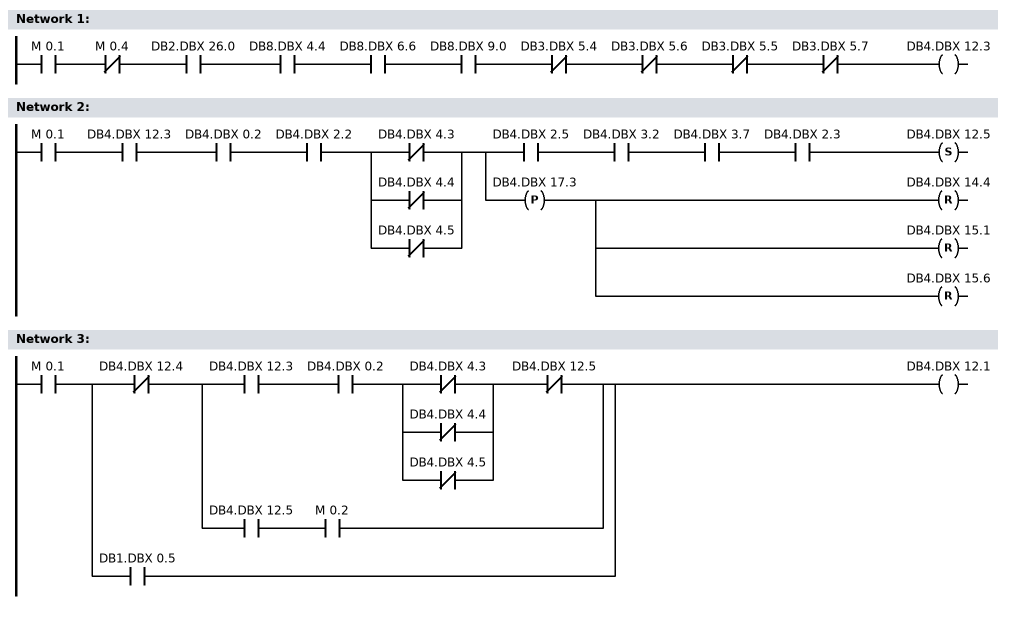
NETWORK
TITLE =
      A     M 0.1;
      AN    M 0.4;
      A     DB2.DBX 26.0;
      A     DB8.DBX 4.4;
      A     DB8.DBX 6.6;
      A     DB8.DBX 9.0;
      AN    DB3.DBX 5.4;
      AN    DB3.DBX 5.6;
      AN    DB3.DBX 5.5;
      AN    DB3.DBX 5.7;
      =     DB4.DBX 12.3;
NETWORK
TITLE =
      A     M 0.1;
      A     DB4.DBX 12.3;
      A     DB4.DBX 0.2;
      A     DB4.DBX 2.2;
      A(;
      ON    DB4.DBX 4.3;
      ON    DB4.DBX 4.4;
      ON    DB4.DBX 4.5;
      );
      =     L 0.0;
      A     L 0.0;
      A     DB4.DBX 2.5;
      A     DB4.DBX 3.2;
      A     DB4.DBX 3.7;
      A     DB4.DBX 2.3;
      S     DB4.DBX 12.5;
      A     L 0.0;
      FP    DB4.DBX 17.3;
      R     DB4.DBX 14.4;
      R     DB4.DBX 15.1;
      R     DB4.DBX 15.6;
NETWORK
TITLE =
      A     M 0.1;
      A(;
      AN    DB4.DBX 12.4;
      A(;
      A     DB4.DBX 12.3;
      A     DB4.DBX 0.2;
      A(;
      ON    DB4.DBX 4.3;
      ON    DB4.DBX 4.4;
      ON    DB4.DBX 4.5;
      );
      AN    DB4.DBX 12.5;
      O;
      A     DB4.DBX 12.5;
      A     M 0.2;
      );
      O     DB1.DBX 0.5;
      );
      =     DB4.DBX 12.1;
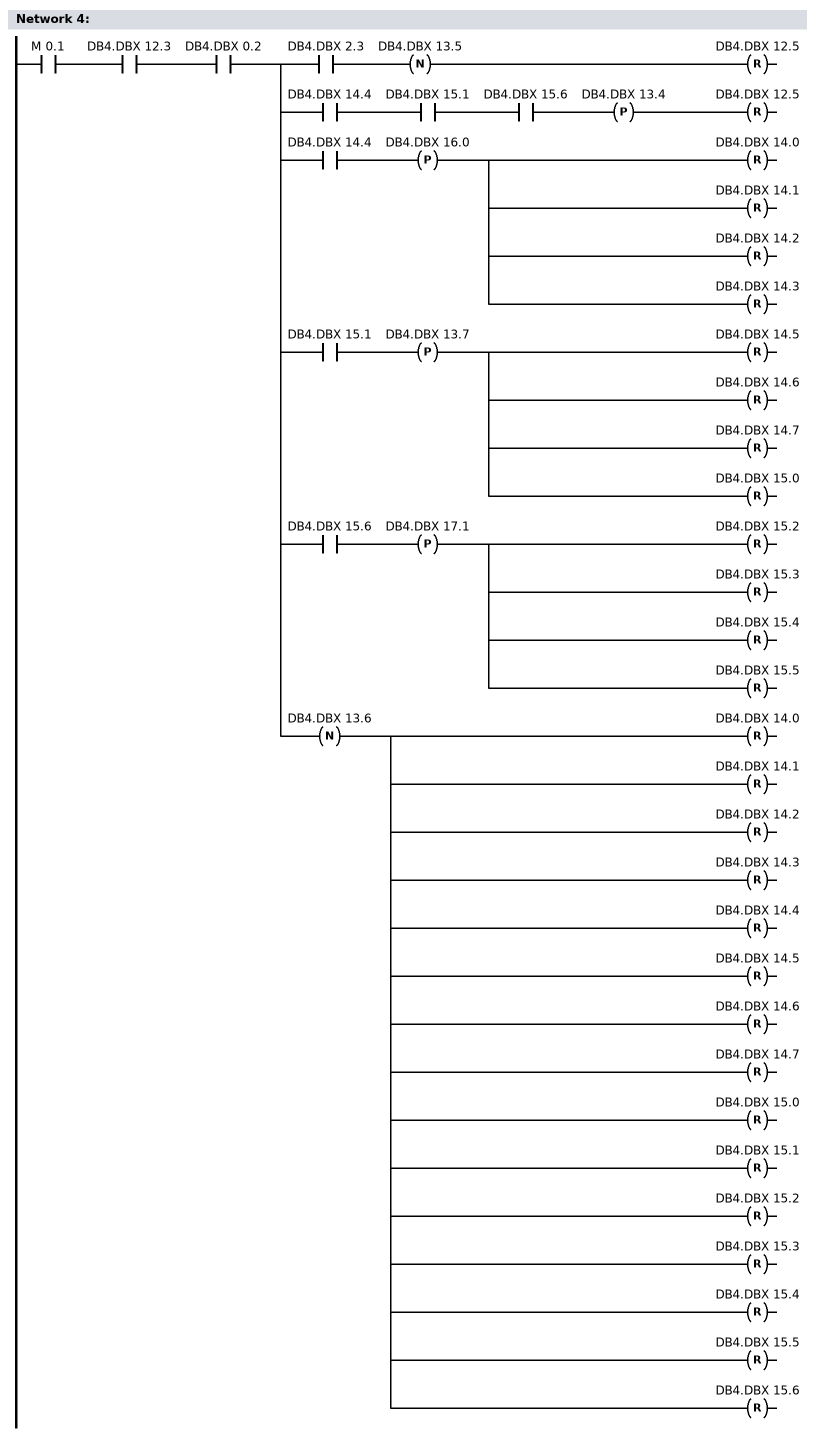
NETWORK
TITLE =
      A     M 0.1;
      A     DB4.DBX 12.3;
      A     DB4.DBX 0.2;
      =     L 0.0;
      A     L 0.0;
      A     DB4.DBX 2.3;
      FN    DB4.DBX 13.5;
      R     DB4.DBX 12.5;
      A     L 0.0;
      A     DB4.DBX 14.4;
      A     DB4.DBX 15.1;
      A     DB4.DBX 15.6;
      FP    DB4.DBX 13.4;
      R     DB4.DBX 12.5;
      A     L 0.0;
      A     DB4.DBX 14.4;
      FP    DB4.DBX 16.0;
      R     DB4.DBX 14.0;
      R     DB4.DBX 14.1;
      R     DB4.DBX 14.2;
      R     DB4.DBX 14.3;
      A     L 0.0;
      A     DB4.DBX 15.1;
      FP    DB4.DBX 13.7;
      R     DB4.DBX 14.5;
      R     DB4.DBX 14.6;
      R     DB4.DBX 14.7;
      R     DB4.DBX 15.0;
      A     L 0.0;
      A     DB4.DBX 15.6;
      FP    DB4.DBX 17.1;
      R     DB4.DBX 15.2;
      R     DB4.DBX 15.3;
      R     DB4.DBX 15.4;
      R     DB4.DBX 15.5;
      A     L 0.0;
      FN    DB4.DBX 13.6;
      R     DB4.DBX 14.0;
      R     DB4.DBX 14.1;
      R     DB4.DBX 14.2;
      R     DB4.DBX 14.3;
      R     DB4.DBX 14.4;
      R     DB4.DBX 14.5;
      R     DB4.DBX 14.6;
      R     DB4.DBX 14.7;
      R     DB4.DBX 15.0;
      R     DB4.DBX 15.1;
      R     DB4.DBX 15.2;
      R     DB4.DBX 15.3;
      R     DB4.DBX 15.4;
      R     DB4.DBX 15.5;
      R     DB4.DBX 15.6;
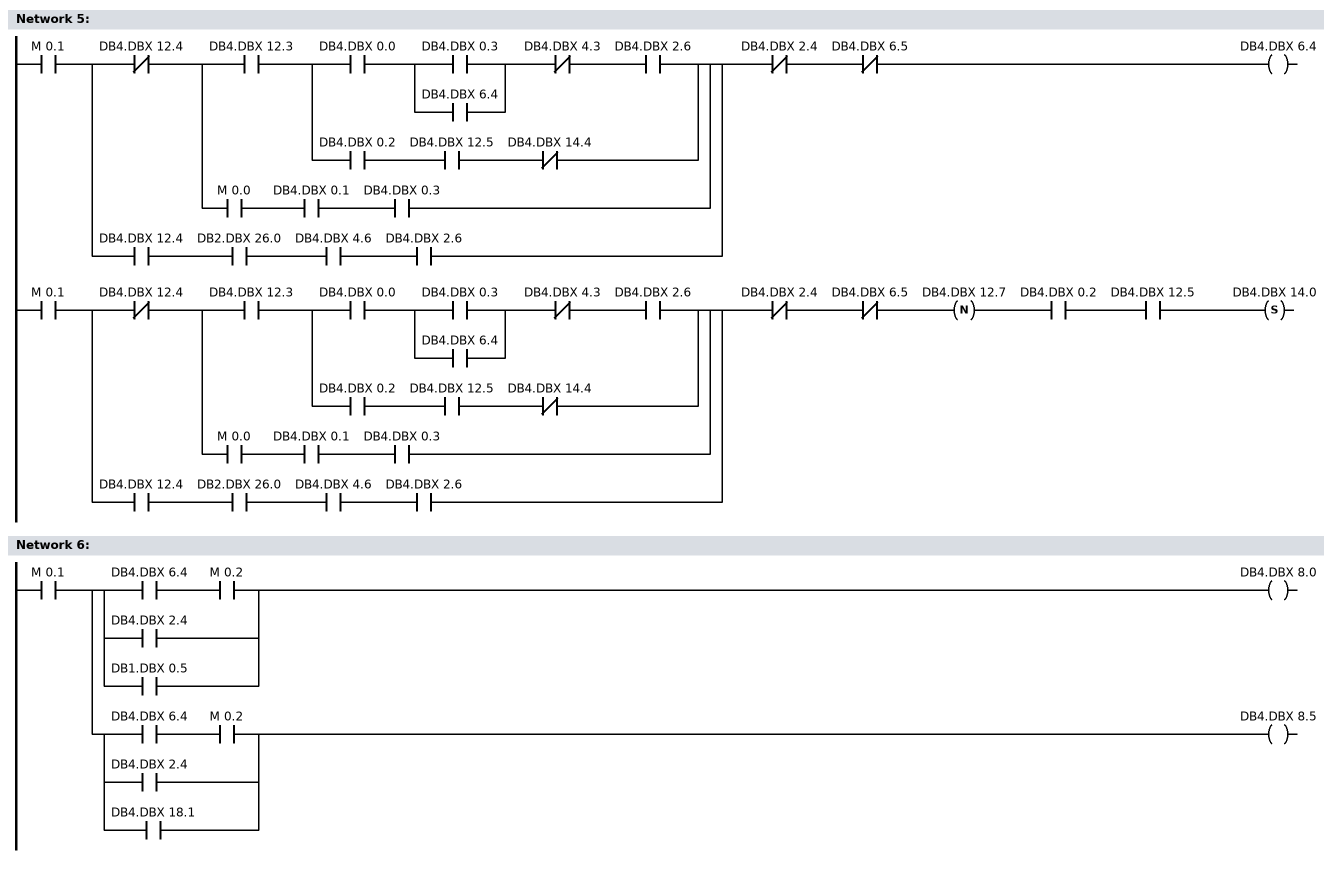
NETWORK
TITLE =
      A     M 0.1;
      A(;
      AN    DB4.DBX 12.4;
      A(;
      A     DB4.DBX 12.3;
      A(;
      A     DB4.DBX 0.0;
      A(;
      O     DB4.DBX 0.3;
      O     DB4.DBX 6.4;
      );
      AN    DB4.DBX 4.3;
      A     DB4.DBX 2.6;
      O;
      A     DB4.DBX 0.2;
      A     DB4.DBX 12.5;
      AN    DB4.DBX 14.4;
      );
      O;
      A     M 0.0;
      A     DB4.DBX 0.1;
      A     DB4.DBX 0.3;
      );
      O;
      A     DB4.DBX 12.4;
      A     DB2.DBX 26.0;
      A     DB4.DBX 4.6;
      A     DB4.DBX 2.6;
      );
      AN    DB4.DBX 2.4;
      AN    DB4.DBX 6.5;
      =     L 0.0;
      A     L 0.0;
      BLD   102;
      =     DB4.DBX 6.4;
      A(;
      A     L 0.0;
      FN    DB4.DBX 12.7;
      );
      A     DB4.DBX 0.2;
      A     DB4.DBX 12.5;
      S     DB4.DBX 14.0;
NETWORK
TITLE =
      A     M 0.1;
      =     L 0.0;
      A     L 0.0;
      A(;
      A     DB4.DBX 6.4;
      A     M 0.2;
      O     DB4.DBX 2.4;
      O     DB1.DBX 0.5;
      );
      =     DB4.DBX 8.0;
      A     L 0.0;
      A(;
      A     DB4.DBX 6.4;
      A     M 0.2;
      O     DB4.DBX 2.4;
      O     DB4.DBX 18.1;
      );
      =     DB4.DBX 8.5;
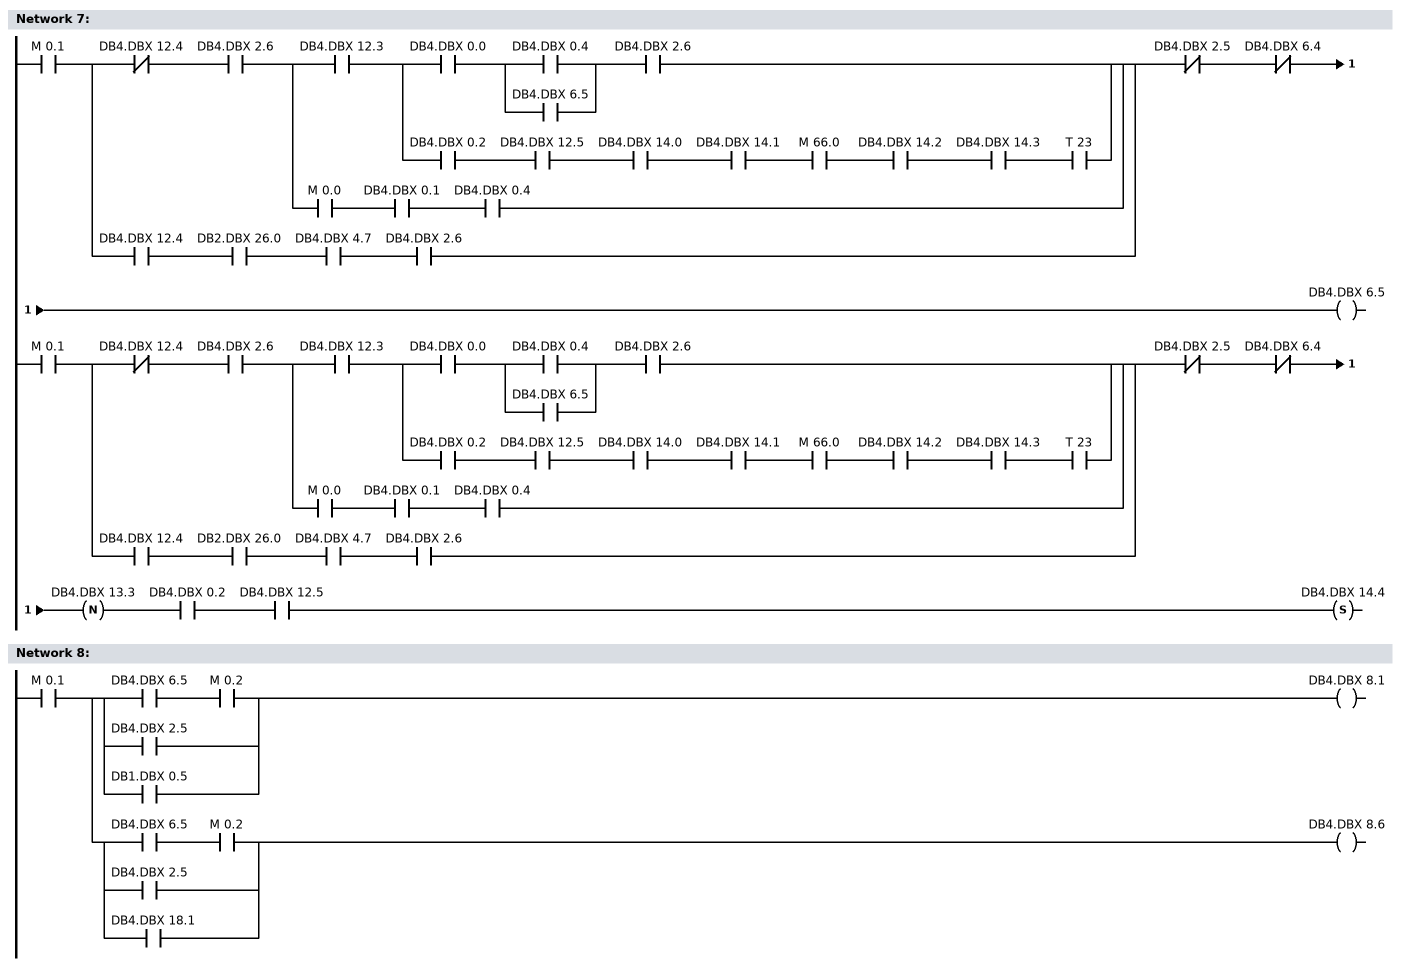
NETWORK
TITLE =
      A     M 0.1;
      A(;
      AN    DB4.DBX 12.4;
      A     DB4.DBX 2.6;
      A(;
      A     DB4.DBX 12.3;
      A(;
      A     DB4.DBX 0.0;
      A(;
      O     DB4.DBX 0.4;
      O     DB4.DBX 6.5;
      );
      A     DB4.DBX 2.6;
      O;
      A     DB4.DBX 0.2;
      A     DB4.DBX 12.5;
      A     DB4.DBX 14.0;
      A     DB4.DBX 14.1;
      A     M 66.0;
      A     DB4.DBX 14.2;
      A     DB4.DBX 14.3;
      A     T 23;
      );
      O;
      A     M 0.0;
      A     DB4.DBX 0.1;
      A     DB4.DBX 0.4;
      );
      O;
      A     DB4.DBX 12.4;
      A     DB2.DBX 26.0;
      A     DB4.DBX 4.7;
      A     DB4.DBX 2.6;
      );
      AN    DB4.DBX 2.5;
      AN    DB4.DBX 6.4;
      =     L 0.0;
      A     L 0.0;
      BLD   102;
      =     DB4.DBX 6.5;
      A(;
      A     L 0.0;
      FN    DB4.DBX 13.3;
      );
      A     DB4.DBX 0.2;
      A     DB4.DBX 12.5;
      S     DB4.DBX 14.4;
NETWORK
TITLE =
      A     M 0.1;
      =     L 0.0;
      A     L 0.0;
      A(;
      A     DB4.DBX 6.5;
      A     M 0.2;
      O     DB4.DBX 2.5;
      O     DB1.DBX 0.5;
      );
      =     DB4.DBX 8.1;
      A     L 0.0;
      A(;
      A     DB4.DBX 6.5;
      A     M 0.2;
      O     DB4.DBX 2.5;
      O     DB4.DBX 18.1;
      );
      =     DB4.DBX 8.6;
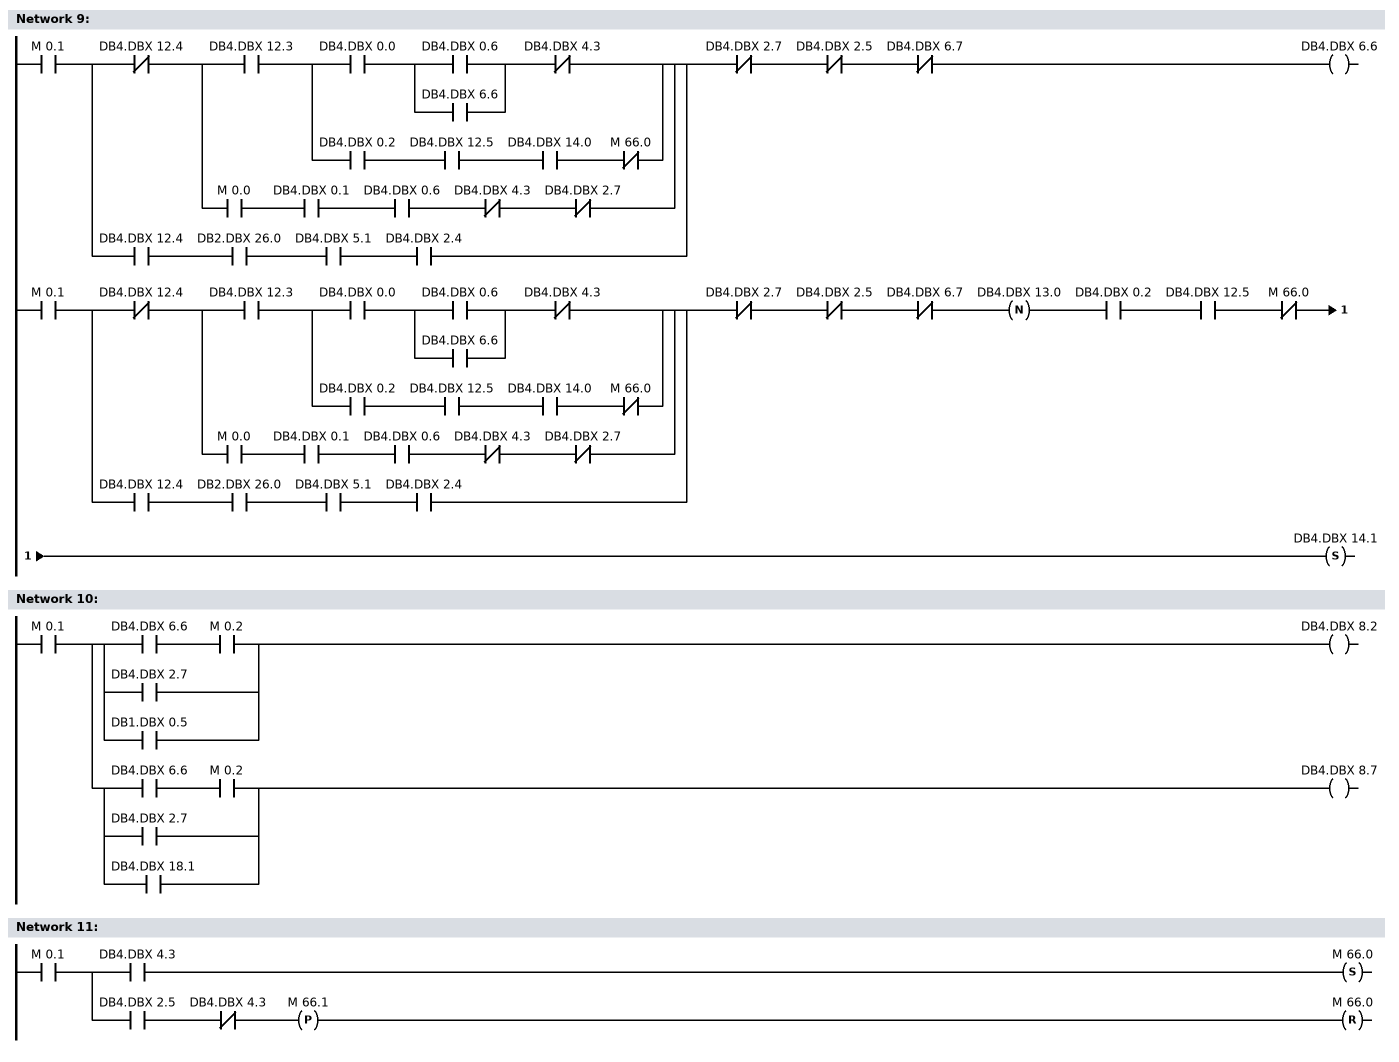
NETWORK
TITLE =
      A     M 0.1;
      A(;
      AN    DB4.DBX 12.4;
      A(;
      A     DB4.DBX 12.3;
      A(;
      A     DB4.DBX 0.0;
      A(;
      O     DB4.DBX 0.6;
      O     DB4.DBX 6.6;
      );
      AN    DB4.DBX 4.3;
      O;
      A     DB4.DBX 0.2;
      A     DB4.DBX 12.5;
      A     DB4.DBX 14.0;
      AN    M 66.0;
      );
      O;
      A     M 0.0;
      A     DB4.DBX 0.1;
      A     DB4.DBX 0.6;
      AN    DB4.DBX 4.3;
      AN    DB4.DBX 2.7;
      );
      O;
      A     DB4.DBX 12.4;
      A     DB2.DBX 26.0;
      A     DB4.DBX 5.1;
      A     DB4.DBX 2.4;
      );
      AN    DB4.DBX 2.7;
      AN    DB4.DBX 2.5;
      AN    DB4.DBX 6.7;
      =     L 0.0;
      A     L 0.0;
      BLD   102;
      =     DB4.DBX 6.6;
      A(;
      A     L 0.0;
      FN    DB4.DBX 13.0;
      );
      A     DB4.DBX 0.2;
      A     DB4.DBX 12.5;
      AN    M 66.0;
      S     DB4.DBX 14.1;
NETWORK
TITLE =
      A     M 0.1;
      =     L 0.0;
      A     L 0.0;
      A(;
      A     DB4.DBX 6.6;
      A     M 0.2;
      O     DB4.DBX 2.7;
      O     DB1.DBX 0.5;
      );
      =     DB4.DBX 8.2;
      A     L 0.0;
      A(;
      A     DB4.DBX 6.6;
      A     M 0.2;
      O     DB4.DBX 2.7;
      O     DB4.DBX 18.1;
      );
      =     DB4.DBX 8.7;
NETWORK
TITLE =
      A     M 0.1;
      =     L 0.0;
      A     L 0.0;
      A     DB4.DBX 4.3;
      S     M 66.0;
      A     L 0.0;
      A     DB4.DBX 2.5;
      AN    DB4.DBX 4.3;
      FP    M 66.1;
      R     M 66.0;
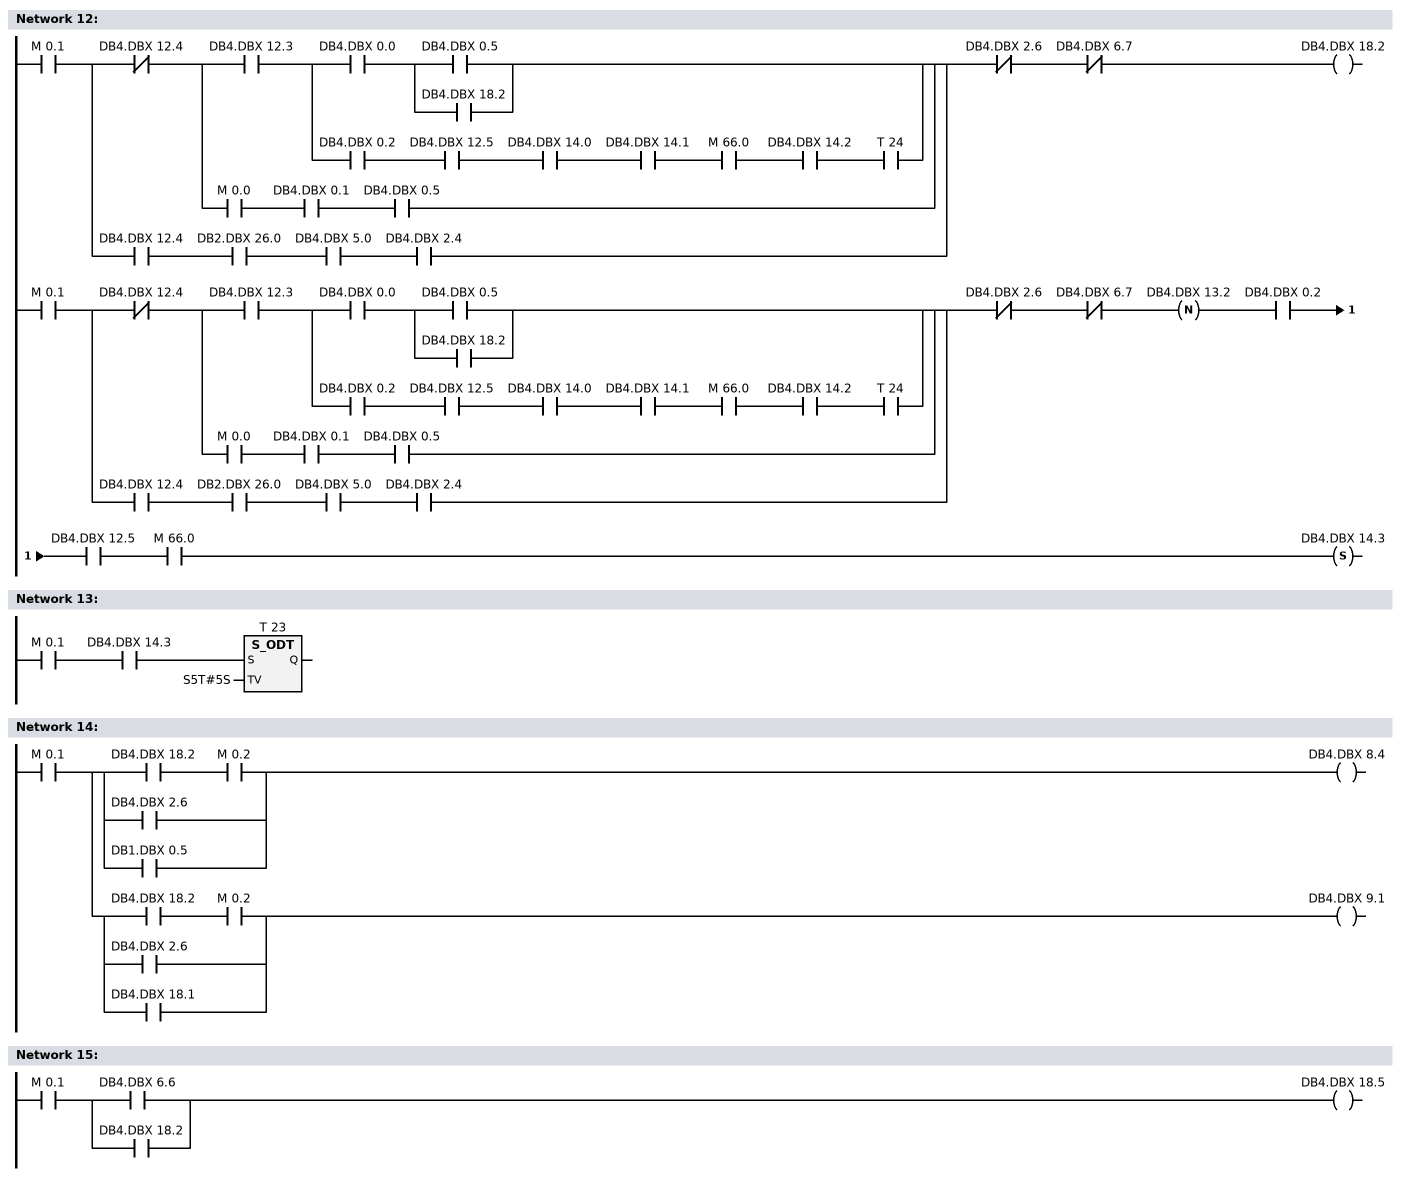
NETWORK
TITLE =
      A     M 0.1;
      A(;
      AN    DB4.DBX 12.4;
      A(;
      A     DB4.DBX 12.3;
      A(;
      A     DB4.DBX 0.0;
      A(;
      O     DB4.DBX 0.5;
      O     DB4.DBX 18.2;
      );
      O;
      A     DB4.DBX 0.2;
      A     DB4.DBX 12.5;
      A     DB4.DBX 14.0;
      A     DB4.DBX 14.1;
      A     M 66.0;
      A     DB4.DBX 14.2;
      A     T 24;
      );
      O;
      A     M 0.0;
      A     DB4.DBX 0.1;
      A     DB4.DBX 0.5;
      );
      O;
      A     DB4.DBX 12.4;
      A     DB2.DBX 26.0;
      A     DB4.DBX 5.0;
      A     DB4.DBX 2.4;
      );
      AN    DB4.DBX 2.6;
      AN    DB4.DBX 6.7;
      =     L 0.0;
      A     L 0.0;
      BLD   102;
      =     DB4.DBX 18.2;
      A(;
      A     L 0.0;
      FN    DB4.DBX 13.2;
      );
      A     DB4.DBX 0.2;
      A     DB4.DBX 12.5;
      A     M 66.0;
      S     DB4.DBX 14.3;
NETWORK
TITLE =
      A     M 0.1;
      A     DB4.DBX 14.3;
      L     S5T#5S;
      SD    T 23;
      NOP   0;
      NOP   0;
      NOP   0;
      NOP   0;
NETWORK
TITLE =
      A     M 0.1;
      =     L 0.0;
      A     L 0.0;
      A(;
      A     DB4.DBX 18.2;
      A     M 0.2;
      O     DB4.DBX 2.6;
      O     DB1.DBX 0.5;
      );
      =     DB4.DBX 8.4;
      A     L 0.0;
      A(;
      A     DB4.DBX 18.2;
      A     M 0.2;
      O     DB4.DBX 2.6;
      O     DB4.DBX 18.1;
      );
      =     DB4.DBX 9.1;
NETWORK
TITLE =
      A     M 0.1;
      A(;
      O     DB4.DBX 6.6;
      O     DB4.DBX 18.2;
      );
      =     DB4.DBX 18.5;
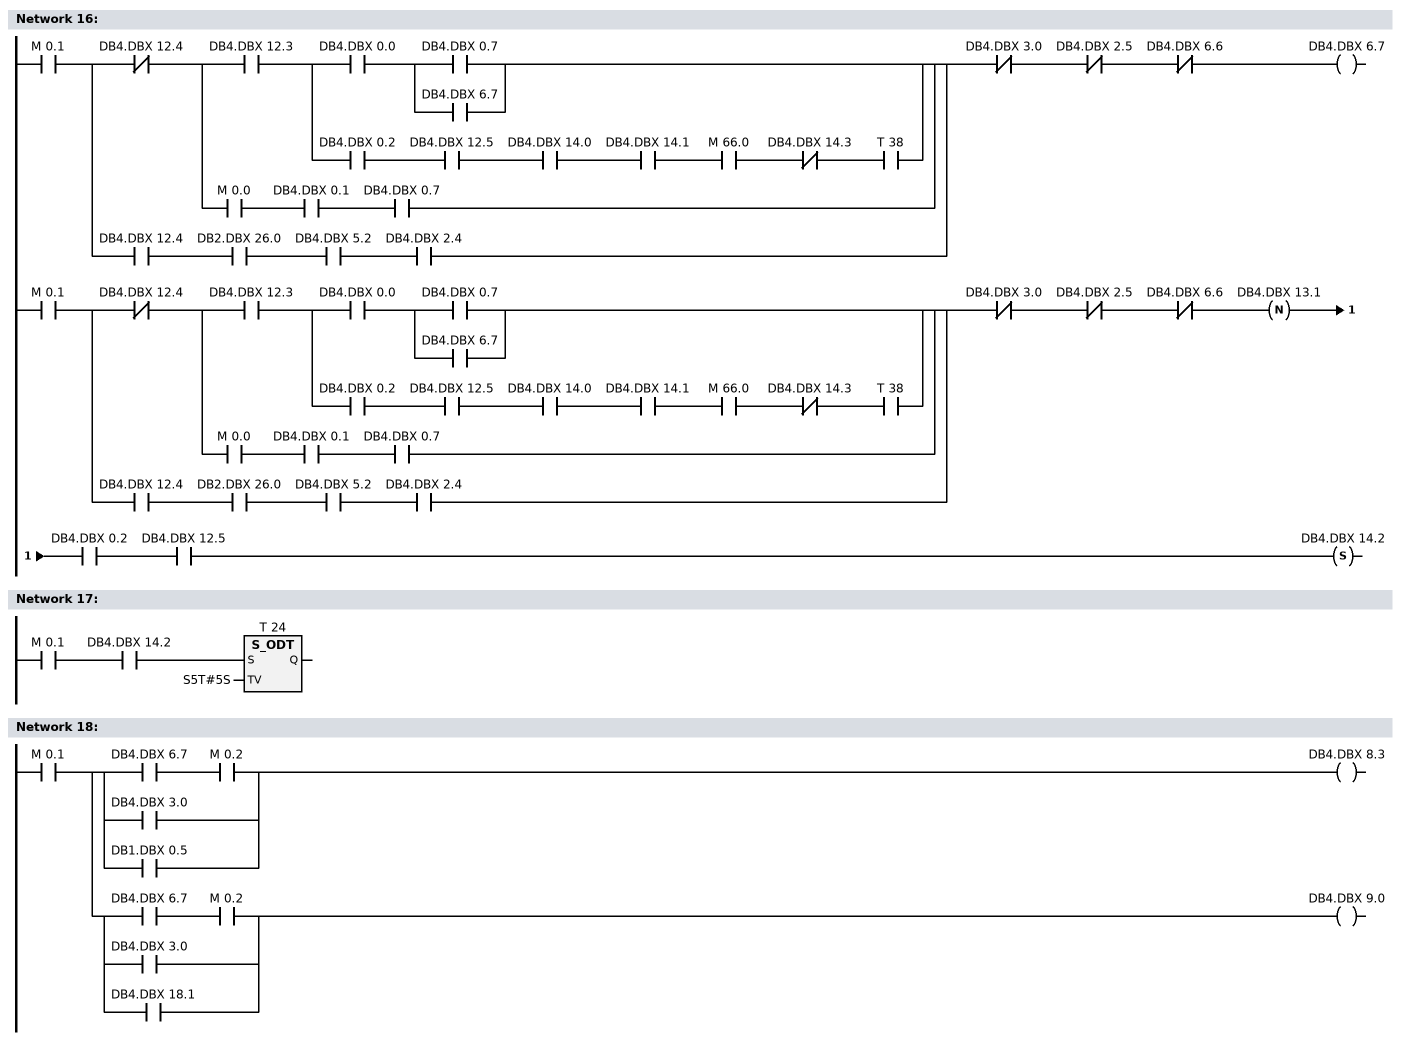
NETWORK
TITLE =
      A     M 0.1;
      A(;
      AN    DB4.DBX 12.4;
      A(;
      A     DB4.DBX 12.3;
      A(;
      A     DB4.DBX 0.0;
      A(;
      O     DB4.DBX 0.7;
      O     DB4.DBX 6.7;
      );
      O;
      A     DB4.DBX 0.2;
      A     DB4.DBX 12.5;
      A     DB4.DBX 14.0;
      A     DB4.DBX 14.1;
      A     M 66.0;
      AN    DB4.DBX 14.3;
      A     T 38;
      );
      O;
      A     M 0.0;
      A     DB4.DBX 0.1;
      A     DB4.DBX 0.7;
      );
      O;
      A     DB4.DBX 12.4;
      A     DB2.DBX 26.0;
      A     DB4.DBX 5.2;
      A     DB4.DBX 2.4;
      );
      AN    DB4.DBX 3.0;
      AN    DB4.DBX 2.5;
      AN    DB4.DBX 6.6;
      =     L 0.0;
      A     L 0.0;
      BLD   102;
      =     DB4.DBX 6.7;
      A(;
      A     L 0.0;
      FN    DB4.DBX 13.1;
      );
      A     DB4.DBX 0.2;
      A     DB4.DBX 12.5;
      S     DB4.DBX 14.2;
NETWORK
TITLE =
      A     M 0.1;
      A     DB4.DBX 14.2;
      L     S5T#5S;
      SD    T 24;
      NOP   0;
      NOP   0;
      NOP   0;
      NOP   0;
NETWORK
TITLE =
      A     M 0.1;
      =     L 0.0;
      A     L 0.0;
      A(;
      A     DB4.DBX 6.7;
      A     M 0.2;
      O     DB4.DBX 3.0;
      O     DB1.DBX 0.5;
      );
      =     DB4.DBX 8.3;
      A     L 0.0;
      A(;
      A     DB4.DBX 6.7;
      A     M 0.2;
      O     DB4.DBX 3.0;
      O     DB4.DBX 18.1;
      );
      =     DB4.DBX 9.0;
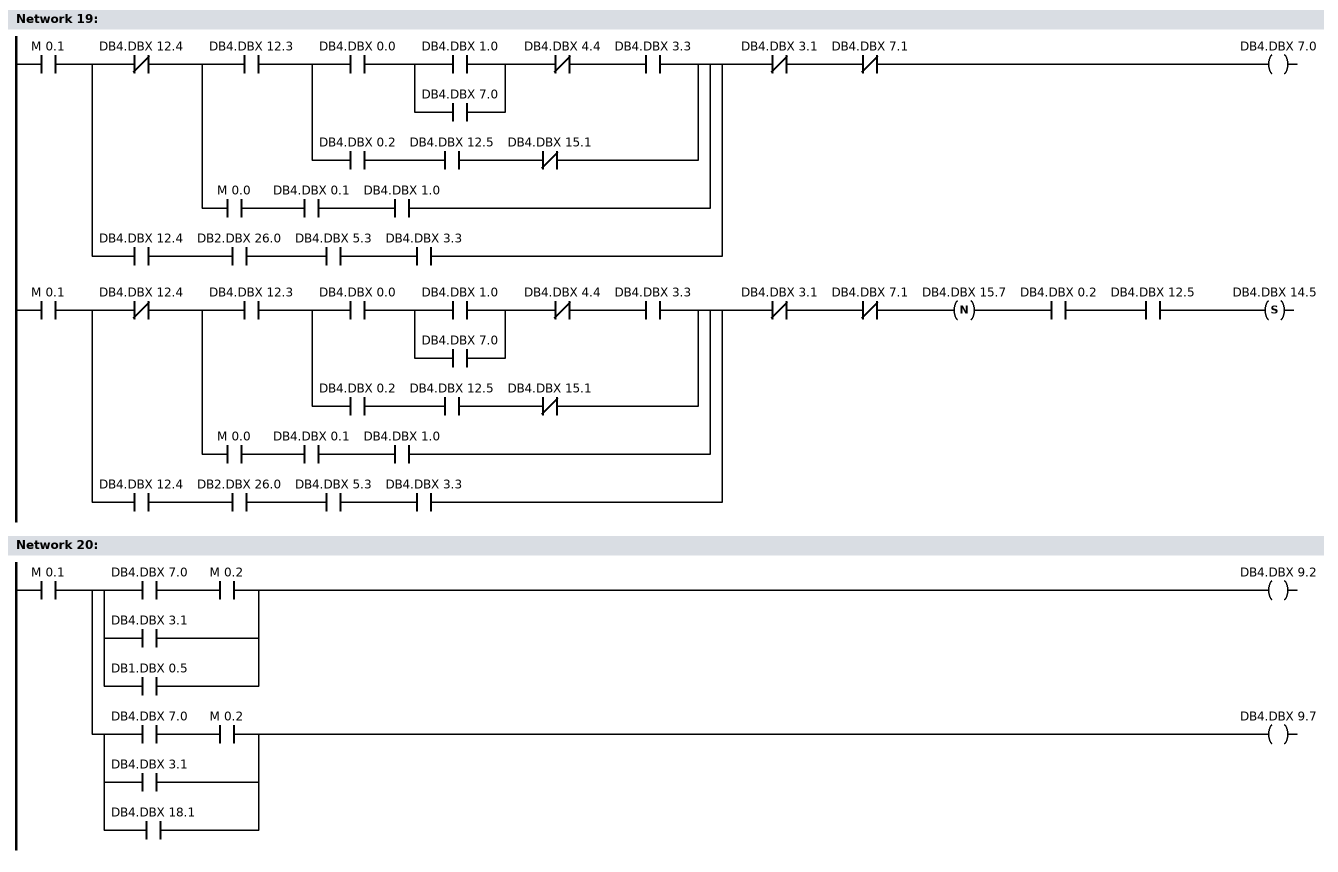
NETWORK
TITLE =
      A     M 0.1;
      A(;
      AN    DB4.DBX 12.4;
      A(;
      A     DB4.DBX 12.3;
      A(;
      A     DB4.DBX 0.0;
      A(;
      O     DB4.DBX 1.0;
      O     DB4.DBX 7.0;
      );
      AN    DB4.DBX 4.4;
      A     DB4.DBX 3.3;
      O;
      A     DB4.DBX 0.2;
      A     DB4.DBX 12.5;
      AN    DB4.DBX 15.1;
      );
      O;
      A     M 0.0;
      A     DB4.DBX 0.1;
      A     DB4.DBX 1.0;
      );
      O;
      A     DB4.DBX 12.4;
      A     DB2.DBX 26.0;
      A     DB4.DBX 5.3;
      A     DB4.DBX 3.3;
      );
      AN    DB4.DBX 3.1;
      AN    DB4.DBX 7.1;
      =     L 0.0;
      A     L 0.0;
      BLD   102;
      =     DB4.DBX 7.0;
      A(;
      A     L 0.0;
      FN    DB4.DBX 15.7;
      );
      A     DB4.DBX 0.2;
      A     DB4.DBX 12.5;
      S     DB4.DBX 14.5;
NETWORK
TITLE =
      A     M 0.1;
      =     L 0.0;
      A     L 0.0;
      A(;
      A     DB4.DBX 7.0;
      A     M 0.2;
      O     DB4.DBX 3.1;
      O     DB1.DBX 0.5;
      );
      =     DB4.DBX 9.2;
      A     L 0.0;
      A(;
      A     DB4.DBX 7.0;
      A     M 0.2;
      O     DB4.DBX 3.1;
      O     DB4.DBX 18.1;
      );
      =     DB4.DBX 9.7;
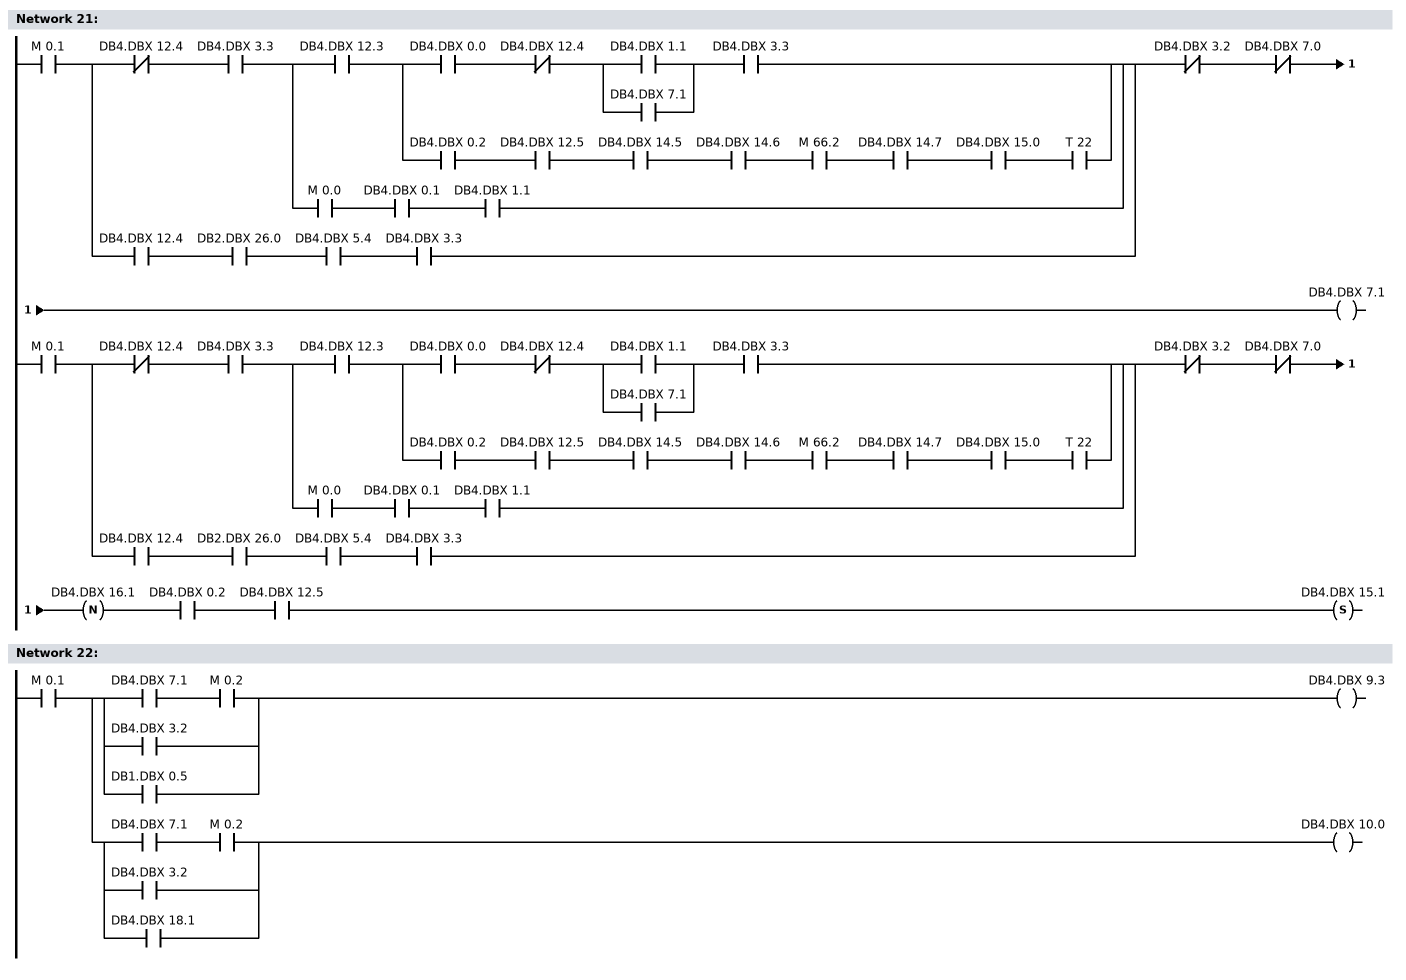
NETWORK
TITLE =
      A     M 0.1;
      A(;
      AN    DB4.DBX 12.4;
      A     DB4.DBX 3.3;
      A(;
      A     DB4.DBX 12.3;
      A(;
      A     DB4.DBX 0.0;
      AN    DB4.DBX 12.4;
      A(;
      O     DB4.DBX 1.1;
      O     DB4.DBX 7.1;
      );
      A     DB4.DBX 3.3;
      O;
      A     DB4.DBX 0.2;
      A     DB4.DBX 12.5;
      A     DB4.DBX 14.5;
      A     DB4.DBX 14.6;
      A     M 66.2;
      A     DB4.DBX 14.7;
      A     DB4.DBX 15.0;
      A     T 22;
      );
      O;
      A     M 0.0;
      A     DB4.DBX 0.1;
      A     DB4.DBX 1.1;
      );
      O;
      A     DB4.DBX 12.4;
      A     DB2.DBX 26.0;
      A     DB4.DBX 5.4;
      A     DB4.DBX 3.3;
      );
      AN    DB4.DBX 3.2;
      AN    DB4.DBX 7.0;
      =     L 0.0;
      A     L 0.0;
      BLD   102;
      =     DB4.DBX 7.1;
      A(;
      A     L 0.0;
      FN    DB4.DBX 16.1;
      );
      A     DB4.DBX 0.2;
      A     DB4.DBX 12.5;
      S     DB4.DBX 15.1;
NETWORK
TITLE =
      A     M 0.1;
      =     L 0.0;
      A     L 0.0;
      A(;
      A     DB4.DBX 7.1;
      A     M 0.2;
      O     DB4.DBX 3.2;
      O     DB1.DBX 0.5;
      );
      =     DB4.DBX 9.3;
      A     L 0.0;
      A(;
      A     DB4.DBX 7.1;
      A     M 0.2;
      O     DB4.DBX 3.2;
      O     DB4.DBX 18.1;
      );
      =     DB4.DBX 10.0;
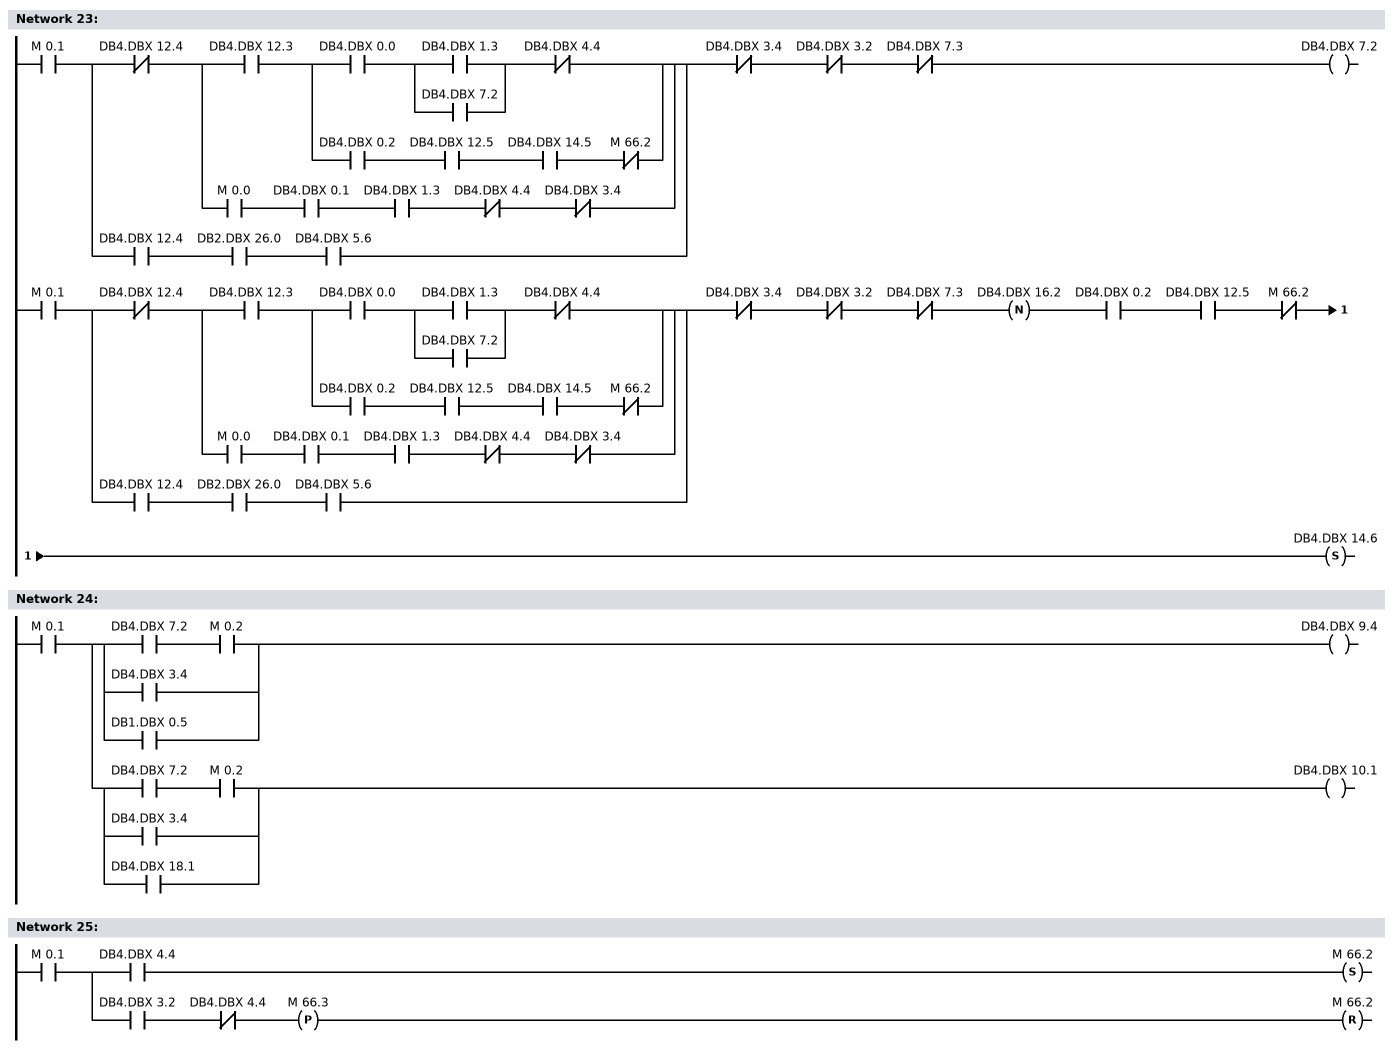
NETWORK
TITLE =
      A     M 0.1;
      A(;
      AN    DB4.DBX 12.4;
      A(;
      A     DB4.DBX 12.3;
      A(;
      A     DB4.DBX 0.0;
      A(;
      O     DB4.DBX 1.3;
      O     DB4.DBX 7.2;
      );
      AN    DB4.DBX 4.4;
      O;
      A     DB4.DBX 0.2;
      A     DB4.DBX 12.5;
      A     DB4.DBX 14.5;
      AN    M 66.2;
      );
      O;
      A     M 0.0;
      A     DB4.DBX 0.1;
      A     DB4.DBX 1.3;
      AN    DB4.DBX 4.4;
      AN    DB4.DBX 3.4;
      );
      O;
      A     DB4.DBX 12.4;
      A     DB2.DBX 26.0;
      A     DB4.DBX 5.6;
      );
      AN    DB4.DBX 3.4;
      AN    DB4.DBX 3.2;
      AN    DB4.DBX 7.3;
      =     L 0.0;
      A     L 0.0;
      BLD   102;
      =     DB4.DBX 7.2;
      A(;
      A     L 0.0;
      FN    DB4.DBX 16.2;
      );
      A     DB4.DBX 0.2;
      A     DB4.DBX 12.5;
      AN    M 66.2;
      S     DB4.DBX 14.6;
NETWORK
TITLE =
      A     M 0.1;
      =     L 0.0;
      A     L 0.0;
      A(;
      A     DB4.DBX 7.2;
      A     M 0.2;
      O     DB4.DBX 3.4;
      O     DB1.DBX 0.5;
      );
      =     DB4.DBX 9.4;
      A     L 0.0;
      A(;
      A     DB4.DBX 7.2;
      A     M 0.2;
      O     DB4.DBX 3.4;
      O     DB4.DBX 18.1;
      );
      =     DB4.DBX 10.1;
NETWORK
TITLE =
      A     M 0.1;
      =     L 0.0;
      A     L 0.0;
      A     DB4.DBX 4.4;
      S     M 66.2;
      A     L 0.0;
      A     DB4.DBX 3.2;
      AN    DB4.DBX 4.4;
      FP    M 66.3;
      R     M 66.2;
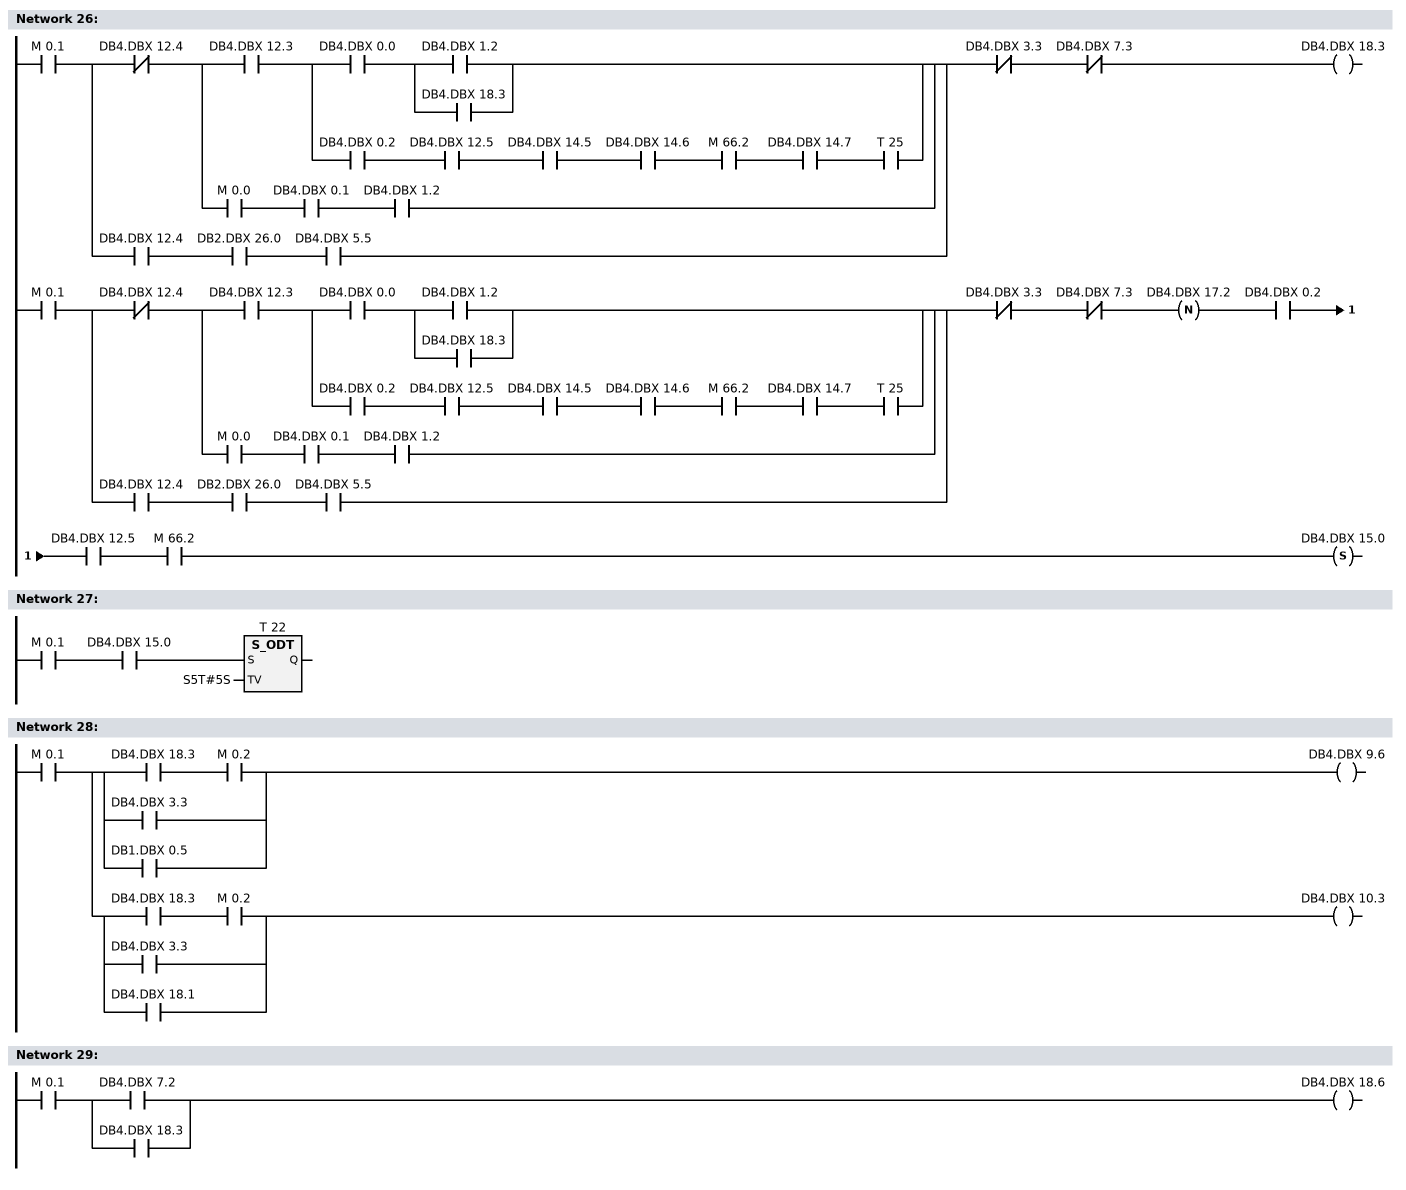
NETWORK
TITLE =
      A     M 0.1;
      A(;
      AN    DB4.DBX 12.4;
      A(;
      A     DB4.DBX 12.3;
      A(;
      A     DB4.DBX 0.0;
      A(;
      O     DB4.DBX 1.2;
      O     DB4.DBX 18.3;
      );
      O;
      A     DB4.DBX 0.2;
      A     DB4.DBX 12.5;
      A     DB4.DBX 14.5;
      A     DB4.DBX 14.6;
      A     M 66.2;
      A     DB4.DBX 14.7;
      A     T 25;
      );
      O;
      A     M 0.0;
      A     DB4.DBX 0.1;
      A     DB4.DBX 1.2;
      );
      O;
      A     DB4.DBX 12.4;
      A     DB2.DBX 26.0;
      A     DB4.DBX 5.5;
      );
      AN    DB4.DBX 3.3;
      AN    DB4.DBX 7.3;
      =     L 0.0;
      A     L 0.0;
      BLD   102;
      =     DB4.DBX 18.3;
      A(;
      A     L 0.0;
      FN    DB4.DBX 17.2;
      );
      A     DB4.DBX 0.2;
      A     DB4.DBX 12.5;
      A     M 66.2;
      S     DB4.DBX 15.0;
NETWORK
TITLE =
      A     M 0.1;
      A     DB4.DBX 15.0;
      L     S5T#5S;
      SD    T 22;
      NOP   0;
      NOP   0;
      NOP   0;
      NOP   0;
NETWORK
TITLE =
      A     M 0.1;
      =     L 0.0;
      A     L 0.0;
      A(;
      A     DB4.DBX 18.3;
      A     M 0.2;
      O     DB4.DBX 3.3;
      O     DB1.DBX 0.5;
      );
      =     DB4.DBX 9.6;
      A     L 0.0;
      A(;
      A     DB4.DBX 18.3;
      A     M 0.2;
      O     DB4.DBX 3.3;
      O     DB4.DBX 18.1;
      );
      =     DB4.DBX 10.3;
NETWORK
TITLE =
      A     M 0.1;
      A(;
      O     DB4.DBX 7.2;
      O     DB4.DBX 18.3;
      );
      =     DB4.DBX 18.6;
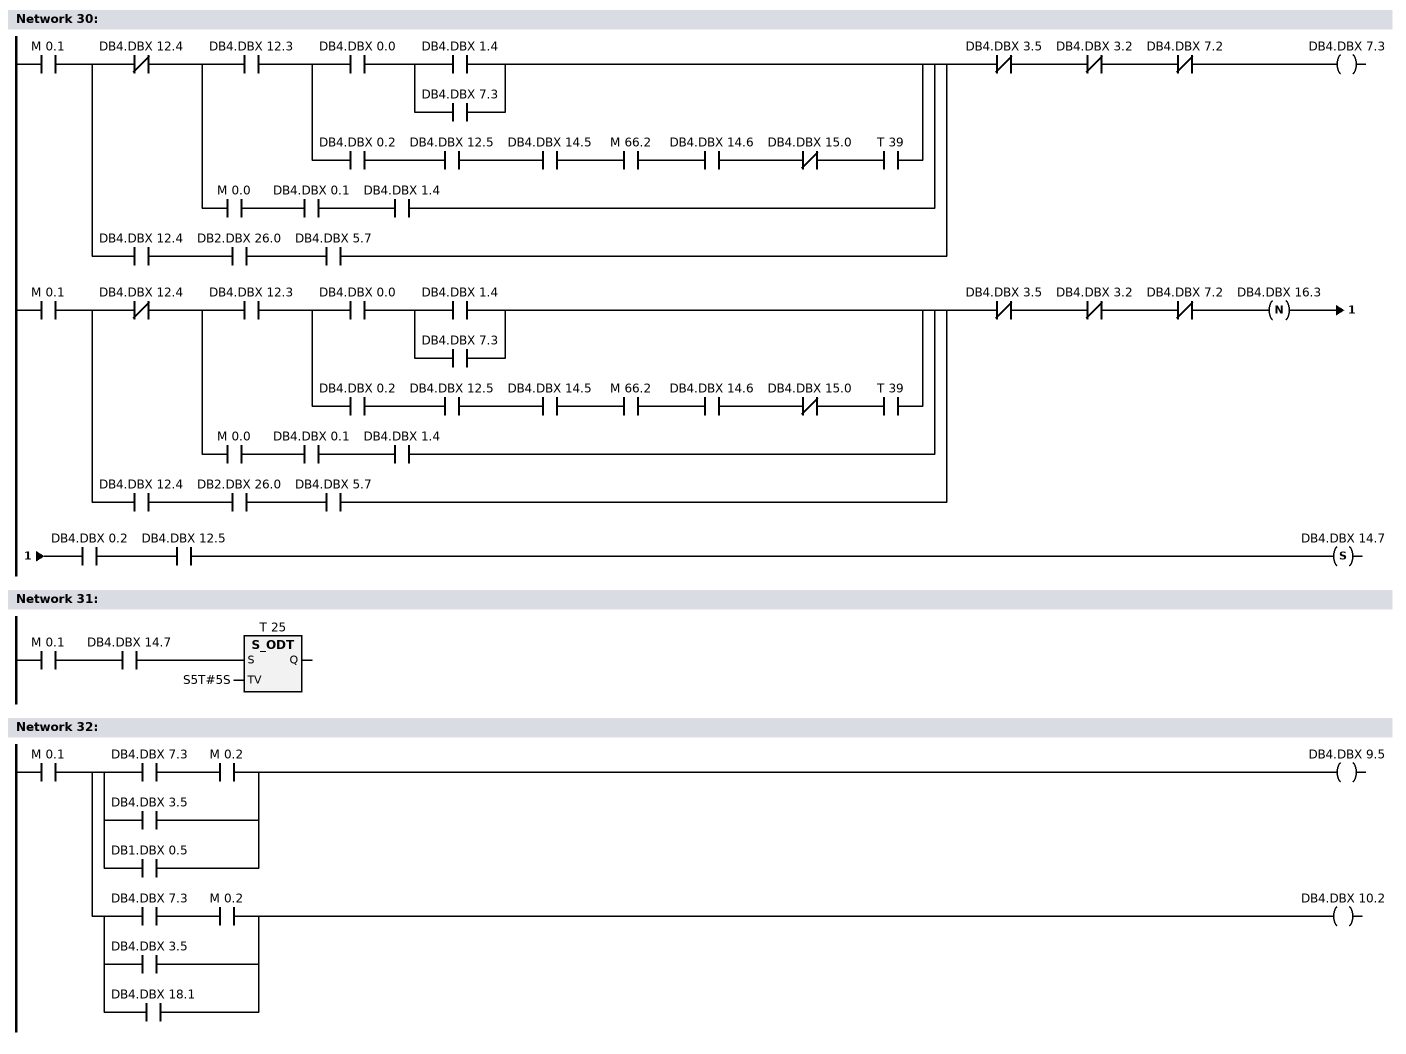
NETWORK
TITLE =
      A     M 0.1;
      A(;
      AN    DB4.DBX 12.4;
      A(;
      A     DB4.DBX 12.3;
      A(;
      A     DB4.DBX 0.0;
      A(;
      O     DB4.DBX 1.4;
      O     DB4.DBX 7.3;
      );
      O;
      A     DB4.DBX 0.2;
      A     DB4.DBX 12.5;
      A     DB4.DBX 14.5;
      A     M 66.2;
      A     DB4.DBX 14.6;
      AN    DB4.DBX 15.0;
      A     T 39;
      );
      O;
      A     M 0.0;
      A     DB4.DBX 0.1;
      A     DB4.DBX 1.4;
      );
      O;
      A     DB4.DBX 12.4;
      A     DB2.DBX 26.0;
      A     DB4.DBX 5.7;
      );
      AN    DB4.DBX 3.5;
      AN    DB4.DBX 3.2;
      AN    DB4.DBX 7.2;
      =     L 0.0;
      A     L 0.0;
      BLD   102;
      =     DB4.DBX 7.3;
      A(;
      A     L 0.0;
      FN    DB4.DBX 16.3;
      );
      A     DB4.DBX 0.2;
      A     DB4.DBX 12.5;
      S     DB4.DBX 14.7;
NETWORK
TITLE =
      A     M 0.1;
      A     DB4.DBX 14.7;
      L     S5T#5S;
      SD    T 25;
      NOP   0;
      NOP   0;
      NOP   0;
      NOP   0;
NETWORK
TITLE =
      A     M 0.1;
      =     L 0.0;
      A     L 0.0;
      A(;
      A     DB4.DBX 7.3;
      A     M 0.2;
      O     DB4.DBX 3.5;
      O     DB1.DBX 0.5;
      );
      =     DB4.DBX 9.5;
      A     L 0.0;
      A(;
      A     DB4.DBX 7.3;
      A     M 0.2;
      O     DB4.DBX 3.5;
      O     DB4.DBX 18.1;
      );
      =     DB4.DBX 10.2;
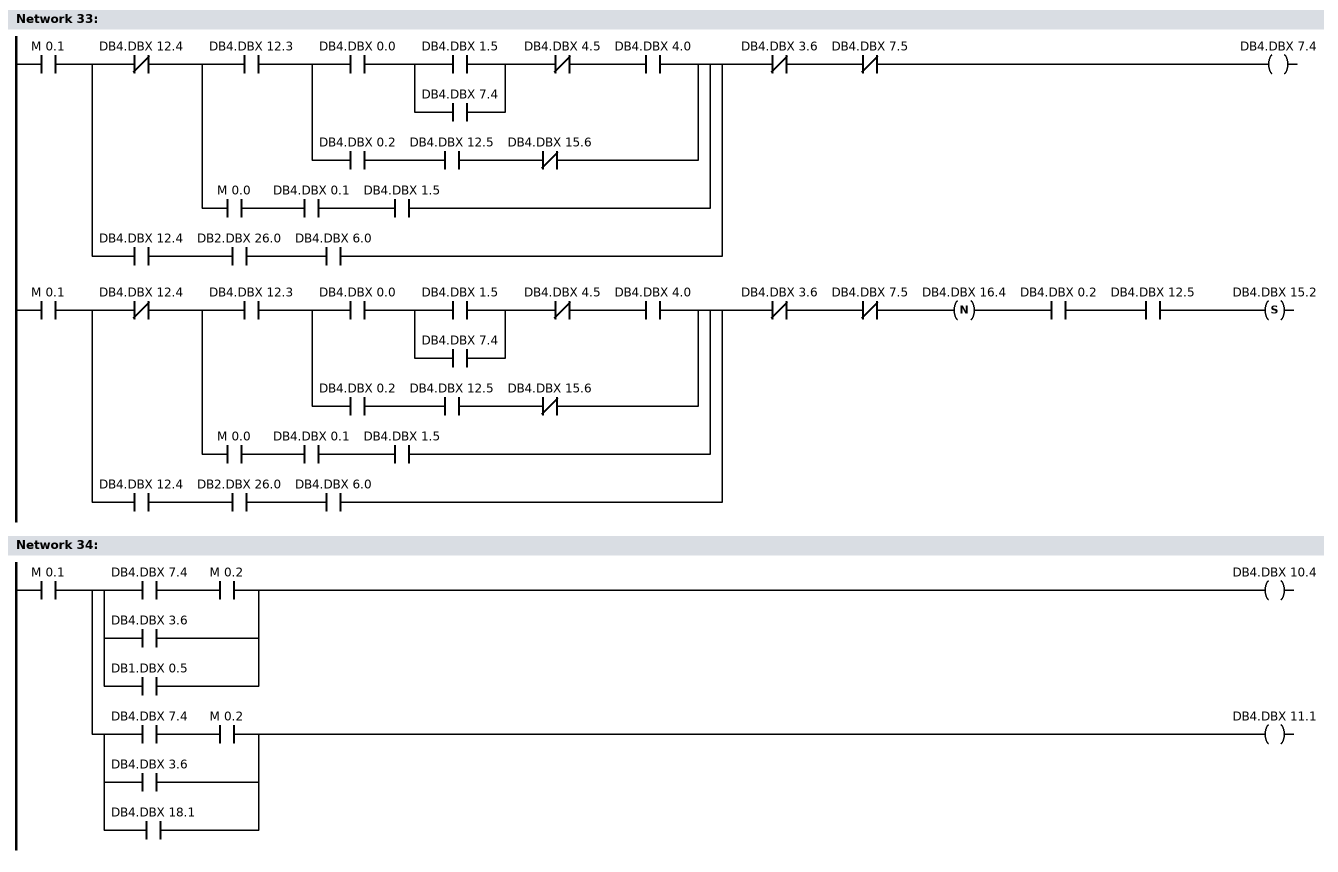
NETWORK
TITLE =
      A     M 0.1;
      A(;
      AN    DB4.DBX 12.4;
      A(;
      A     DB4.DBX 12.3;
      A(;
      A     DB4.DBX 0.0;
      A(;
      O     DB4.DBX 1.5;
      O     DB4.DBX 7.4;
      );
      AN    DB4.DBX 4.5;
      A     DB4.DBX 4.0;
      O;
      A     DB4.DBX 0.2;
      A     DB4.DBX 12.5;
      AN    DB4.DBX 15.6;
      );
      O;
      A     M 0.0;
      A     DB4.DBX 0.1;
      A     DB4.DBX 1.5;
      );
      O;
      A     DB4.DBX 12.4;
      A     DB2.DBX 26.0;
      A     DB4.DBX 6.0;
      );
      AN    DB4.DBX 3.6;
      AN    DB4.DBX 7.5;
      =     L 0.0;
      A     L 0.0;
      BLD   102;
      =     DB4.DBX 7.4;
      A(;
      A     L 0.0;
      FN    DB4.DBX 16.4;
      );
      A     DB4.DBX 0.2;
      A     DB4.DBX 12.5;
      S     DB4.DBX 15.2;
NETWORK
TITLE =
      A     M 0.1;
      =     L 0.0;
      A     L 0.0;
      A(;
      A     DB4.DBX 7.4;
      A     M 0.2;
      O     DB4.DBX 3.6;
      O     DB1.DBX 0.5;
      );
      =     DB4.DBX 10.4;
      A     L 0.0;
      A(;
      A     DB4.DBX 7.4;
      A     M 0.2;
      O     DB4.DBX 3.6;
      O     DB4.DBX 18.1;
      );
      =     DB4.DBX 11.1;
